LIN {X 0,Y 319.606,Z 333.555,A -85,B 0,C 180,E1 -15763.44,E2 -15763.44} C_VEL
LIN {X 0,Y 313.637,Z 316.329,A -85,B 0,C 180,E1 -15764.269,E2 -15764.269} C_VEL
LIN {X 0,Y 312.647,Z 311.538,A -85,B 0,C 180,E1 -15765.774,E2 -15765.774} C_VEL
LIN {X 0,Y 312.557,Z 311.55,A -85,B 0,C 180,E1 -15769.71,E2 -15769.71} C_VEL
LIN {X 0,Y 312.519,Z 311.556,A -85,B 0,C 180,E1 -15772.777,E2 -15772.777} C_VEL
LIN {X 0,Y 312.524,Z 311.552,A -85,B 0,C 180,E1 -15775.906,E2 -15775.906} C_VEL
LIN {X 0,Y 312.491,Z 311.556,A -85,B 0,C 180,E1 -15779.654,E2 -15779.654} C_VEL
LIN {X 0,Y 312.516,Z 311.553,A -85,B 0,C 180,E1 -15783.688,E2 -15783.688} C_VEL
LIN {X 0,Y 312.509,Z 311.554,A -85,B 0,C 180,E1 -15787.386,E2 -15787.386} C_VEL
LIN {X 0,Y 312.422,Z 311.565,A -85,B 0,C 180,E1 -15791.109,E2 -15791.109} C_VEL
LIN {X 0,Y 311.749,Z 311.65,A -85,B 0,C 180,E1 -15792.185,E2 -15792.185} C_VEL
LIN {X 0,Y 308.901,Z 312,A -85,B 0,C 180,E1 -15793.937,E2 -15793.937} C_VEL
LIN {X 0,Y 306.504,Z 312.305,A -85,B 0,C 180,E1 -15795.358,E2 -15795.358} C_VEL
LIN {X 0,Y 305.493,Z 312.428,A -85,B 0,C 180,E1 -15796.458,E2 -15796.458} C_VEL
LIN {X 0,Y 305.42,Z 312.437,A -85,B 0,C 180,E1 -15796.83,E2 -15796.83} C_VEL
LIN {X 0,Y 305.452,Z 312.431,A -85,B 0,C 180,E1 -15799.891,E2 -15799.891} C_VEL
LIN {X 0,Y 305.472,Z 312.433,A -85,B 0,C 180,E1 -15803.632,E2 -15803.632} C_VEL
LIN {X 0,Y 305.459,Z 312.432,A -85,B 0,C 180,E1 -15806.483,E2 -15806.483} C_VEL
LIN {X 0,Y 305.488,Z 312.425,A -85,B 0,C 180,E1 -15810.95,E2 -15810.95} C_VEL
LIN {X 0,Y 305.564,Z 312.421,A -85,B 0,C 180,E1 -15814.087,E2 -15814.087} C_VEL
LIN {X 0,Y 305.474,Z 312.427,A -85,B 0,C 180,E1 -15818.401,E2 -15818.401} C_VEL
LIN {X 0,Y 305.573,Z 312.415,A -85,B 0,C 180,E1 -15821.217,E2 -15821.217} C_VEL
LIN {X 0,Y 305.642,Z 312.411,A -85,B 0,C 180,E1 -15825.349,E2 -15825.349} C_VEL
LIN {X 0,Y 305.627,Z 312.408,A -85,B 0,C 180,E1 -15829.399,E2 -15829.399} C_VEL
LIN {X 0,Y 305.757,Z 312.396,A -85,B 0,C 180,E1 -15832.073,E2 -15832.073} C_VEL
LIN {X 0,Y 305.669,Z 312.408,A -85,B 0,C 180,E1 -15834.723,E2 -15834.723} C_VEL
LIN {X 0,Y 305.948,Z 312.37,A -85,B 0,C 180,E1 -15838.684,E2 -15838.684} C_VEL
LIN {X 0,Y 305.949,Z 312.366,A -85,B 0,C 180,E1 -15841.316,E2 -15841.316} C_VEL
LIN {X 0,Y 305.839,Z 312.389,A -85,B 0,C 180,E1 -15846.598,E2 -15846.598} C_VEL
LIN {X 0,Y 305.729,Z 312.396,A -85,B 0,C 180,E1 -15849.26,E2 -15849.26} C_VEL
LIN {X 0,Y 305.582,Z 312.417,A -85,B 0,C 180,E1 -15853.297,E2 -15853.297} C_VEL
LIN {X 0,Y 305.587,Z 312.417,A -85,B 0,C 180,E1 -15856.021,E2 -15856.021} C_VEL
LIN {X 0,Y 305.57,Z 312.42,A -85,B 0,C 180,E1 -15859.445,E2 -15859.445} C_VEL
LIN {X 0,Y 305.485,Z 312.434,A -85,B 0,C 180,E1 -15863.042,E2 -15863.042} C_VEL
LIN {X 0,Y 305.542,Z 312.422,A -85,B 0,C 180,E1 -15866.228,E2 -15866.228} C_VEL
LIN {X 0,Y 305.492,Z 312.434,A -85,B 0,C 180,E1 -15869.051,E2 -15869.051} C_VEL
LIN {X 0,Y 305.443,Z 312.436,A -85,B 0,C 180,E1 -15871.953,E2 -15871.953} C_VEL
LIN {X 0,Y 305.458,Z 312.438,A -85,B 0,C 180,E1 -15875.114,E2 -15875.114} C_VEL
LIN {X 0,Y 305.463,Z 312.434,A -85,B 0,C 180,E1 -15878.534,E2 -15878.534} C_VEL
LIN {X 0,Y 305.451,Z 312.435,A -85,B 0,C 180,E1 -15882.587,E2 -15882.587} C_VEL
LIN {X 0,Y 305.422,Z 312.438,A -85,B 0,C 180,E1 -15886.346,E2 -15886.346} C_VEL
LIN {X 0,Y 305.455,Z 312.437,A -85,B 0,C 180,E1 -15889.893,E2 -15889.893} C_VEL
LIN {X 0,Y 305.479,Z 312.435,A -85,B 0,C 180,E1 -15893.633,E2 -15893.633} C_VEL
LIN {X 0,Y 305.463,Z 312.435,A -85,B 0,C 180,E1 -15896.484,E2 -15896.484} C_VEL
LIN {X 0,Y 305.466,Z 312.471,A -85,B 0,C 180,E1 -15898.295,E2 -15898.295} C_VEL
LIN {X 0,Y 307.956,Z 324.046,A -85,B 0,C 180,E1 -15901.722,E2 -15901.722} C_VEL
LIN {X 0,Y 309.391,Z 332.337,A -85,B 0,C 180,E1 -15904.071,E2 -15904.071} C_VEL
LIN {X 0,Y 308.836,Z 337.527,A -85,B 0,C 180,E1 -15905.425,E2 -15905.425} C_VEL
LIN {X 0,Y 314.553,Z 379.23,A -85,B 0,C 180,E1 -15906.817,E2 -15906.817} C_VEL
LIN {X 0,Y 313.178,Z 446.148,A -85,B 0,C 180,E1 -15908.355,E2 -15908.355} C_VEL
LIN {X 0,Y 312.374,Z 459.427,A -85,B 0,C 180,E1 -15908.902,E2 -15908.902} C_VEL
LIN {X 0,Y 311.419,Z 472.21,A -85,B 0,C 180,E1 -15909.698,E2 -15909.698} C_VEL
LIN {X 0,Y 310.281,Z 483.534,A -85,B 0,C 180,E1 -15910.656,E2 -15910.656} C_VEL
LIN {X 0,Y 308.964,Z 495.25,A -85,B 0,C 180,E1 -15911.946,E2 -15911.946} C_VEL
LIN {X 0,Y 307.787,Z 505.776,A -85,B 0,C 180,E1 -15913.413,E2 -15913.413} C_VEL
LIN {X 0,Y 306.651,Z 515.269,A -85,B 0,C 180,E1 -15915.059,E2 -15915.059} C_VEL
LIN {X 0,Y 305.483,Z 524.396,A -85,B 0,C 180,E1 -15917.039,E2 -15917.039} C_VEL
LIN {X 0,Y 304.627,Z 531.743,A -85,B 0,C 180,E1 -15919.029,E2 -15919.029} C_VEL
LIN {X 0,Y 304.184,Z 536.708,A -85,B 0,C 180,E1 -15920.693,E2 -15920.693} C_VEL
LIN {X 0,Y 303.825,Z 541.519,A -85,B 0,C 180,E1 -15922.692,E2 -15922.692} C_VEL
LIN {X 0,Y 303.667,Z 545.193,A -85,B 0,C 180,E1 -15924.689,E2 -15924.689} C_VEL
LIN {X 0,Y 303.664,Z 547.088,A -85,B 0,C 180,E1 -15926.019,E2 -15926.019} C_VEL
LIN {X 0,Y 303.644,Z 548.512,A -85,B 0,C 180,E1 -15927.348,E2 -15927.348} C_VEL
LIN {X 0,Y 303.634,Z 549.517,A -85,B 0,C 180,E1 -15928.674,E2 -15928.674} C_VEL
LIN {X 0,Y 303.669,Z 550.131,A -85,B 0,C 180,E1 -15930.001,E2 -15930.001} C_VEL
LIN {X 0,Y 303.607,Z 550.351,A -85,B 0,C 180,E1 -15931.327,E2 -15931.327} C_VEL
LIN {X 0,Y 303.624,Z 550.145,A -85,B 0,C 180,E1 -15932.654,E2 -15932.654} C_VEL
LIN {X 0,Y 303.633,Z 549.536,A -85,B 0,C 180,E1 -15933.982,E2 -15933.982} C_VEL
LIN {X 0,Y 303.661,Z 548.281,A -85,B 0,C 180,E1 -15935.612,E2 -15935.612} C_VEL
LIN {X 0,Y 303.959,Z 545.322,A -85,B 0,C 180,E1 -15937.975,E2 -15937.975} C_VEL
LIN {X 0,Y 304.481,Z 541.759,A -85,B 0,C 180,E1 -15939.97,E2 -15939.97} C_VEL
LIN {X 0,Y 305.288,Z 537.11,A -85,B 0,C 180,E1 -15941.958,E2 -15941.958} C_VEL
LIN {X 0,Y 306.752,Z 530.122,A -85,B 0,C 180,E1 -15944.259,E2 -15944.259} C_VEL
LIN {X 0,Y 308.323,Z 522.727,A -85,B 0,C 180,E1 -15946.179,E2 -15946.179} C_VEL
LIN {X 0,Y 309.752,Z 514.917,A -85,B 0,C 180,E1 -15947.836,E2 -15947.836} C_VEL
LIN {X 0,Y 311.598,Z 505.596,A -85,B 0,C 180,E1 -15949.432,E2 -15949.432} C_VEL
LIN {X 0,Y 313.462,Z 495.268,A -85,B 0,C 180,E1 -15950.851,E2 -15950.851} C_VEL
LIN {X 0,Y 315.387,Z 483.82,A -85,B 0,C 180,E1 -15952.089,E2 -15952.089} C_VEL
LIN {X 0,Y 317.023,Z 471.841,A -85,B 0,C 180,E1 -15953.086,E2 -15953.086} C_VEL
LIN {X 0,Y 318.435,Z 458.547,A -85,B 0,C 180,E1 -15953.882,E2 -15953.882} C_VEL
LIN {X 0,Y 319.456,Z 445.222,A -85,B 0,C 180,E1 -15954.405,E2 -15954.405} C_VEL
LIN {X 0,Y 321.236,Z 381.833,A -85,B 0,C 180,E1 -15955.853,E2 -15955.853} C_VEL
LIN {X 0,Y 318.215,Z 363.674,A -85,B 0,C 180,E1 -15956.623,E2 -15956.623} C_VEL
LIN {X 0,Y 313.97,Z 343.479,A -85,B 0,C 180,E1 -15957.602,E2 -15957.602} C_VEL
LIN {X 0,Y 311.195,Z 336.716,A -85,B 0,C 180,E1 -15958.107,E2 -15958.107} C_VEL
LIN {X 0,Y 309.342,Z 328.013,A -85,B 0,C 180,E1 -15960.837,E2 -15960.837} C_VEL
LIN {X 0,Y 306.721,Z 317.256,A -85,B 0,C 180,E1 -15964.423,E2 -15964.423} C_VEL
LIN {X 0,Y 305.48,Z 312.435,A -85,B 0,C 180,E1 -15966.171,E2 -15966.171} C_VEL
LIN {X 0,Y 305.46,Z 312.434,A -85,B 0,C 180,E1 -15970.108,E2 -15970.108} C_VEL
LIN {X 0,Y 305.427,Z 312.441,A -85,B 0,C 180,E1 -15973.655,E2 -15973.655} C_VEL
LIN {X 0,Y 305.456,Z 312.433,A -85,B 0,C 180,E1 -15977.414,E2 -15977.414} C_VEL
LIN {X 0,Y 305.468,Z 312.433,A -85,B 0,C 180,E1 -15981.596,E2 -15981.596} C_VEL
LIN {X 0,Y 305.463,Z 312.434,A -85,B 0,C 180,E1 -15984.887,E2 -15984.887} C_VEL
LIN {X 0,Y 305.453,Z 312.435,A -85,B 0,C 180,E1 -15988.355,E2 -15988.355} C_VEL
LIN {X 0,Y 305.521,Z 312.428,A -85,B 0,C 180,E1 -15991.114,E2 -15991.114} C_VEL
LIN {X 0,Y 305.572,Z 312.418,A -85,B 0,C 180,E1 -15994.088,E2 -15994.088} C_VEL
LIN {X 0,Y 305.501,Z 312.427,A -85,B 0,C 180,E1 -15998.403,E2 -15998.403} C_VEL
LIN {X 0,Y 305.591,Z 312.412,A -85,B 0,C 180,E1 -16001.217,E2 -16001.217} C_VEL
LIN {X 0,Y 305.649,Z 312.403,A -85,B 0,C 180,E1 -16005.349,E2 -16005.349} C_VEL
LIN {X 0,Y 305.636,Z 312.404,A -85,B 0,C 180,E1 -16009.399,E2 -16009.399} C_VEL
LIN {X 0,Y 305.797,Z 312.39,A -85,B 0,C 180,E1 -16012.074,E2 -16012.074} C_VEL
LIN {X 0,Y 305.686,Z 312.393,A -85,B 0,C 180,E1 -16014.723,E2 -16014.723} C_VEL
LIN {X 0,Y 305.955,Z 312.358,A -85,B 0,C 180,E1 -16018.684,E2 -16018.684} C_VEL
LIN {X 0,Y 305.955,Z 312.368,A -85,B 0,C 180,E1 -16021.316,E2 -16021.316} C_VEL
LIN {X 0,Y 305.849,Z 312.379,A -85,B 0,C 180,E1 -16026.614,E2 -16026.614} C_VEL
LIN {X 0,Y 305.736,Z 312.396,A -85,B 0,C 180,E1 -16029.26,E2 -16029.26} C_VEL
LIN {X 0,Y 305.588,Z 312.415,A -85,B 0,C 180,E1 -16033.296,E2 -16033.296} C_VEL
LIN {X 0,Y 305.594,Z 312.414,A -85,B 0,C 180,E1 -16036.02,E2 -16036.02} C_VEL
LIN {X 0,Y 305.575,Z 312.418,A -85,B 0,C 180,E1 -16039.444,E2 -16039.444} C_VEL
LIN {X 0,Y 305.486,Z 312.431,A -85,B 0,C 180,E1 -16043.039,E2 -16043.039} C_VEL
LIN {X 0,Y 305.531,Z 312.423,A -85,B 0,C 180,E1 -16046.221,E2 -16046.221} C_VEL
LIN {X 0,Y 305.488,Z 312.426,A -85,B 0,C 180,E1 -16049.047,E2 -16049.047} C_VEL
LIN {X 0,Y 305.442,Z 312.429,A -85,B 0,C 180,E1 -16051.952,E2 -16051.952} C_VEL
LIN {X 0,Y 305.462,Z 312.429,A -85,B 0,C 180,E1 -16055.113,E2 -16055.113} C_VEL
LIN {X 0,Y 305.449,Z 312.435,A -85,B 0,C 180,E1 -16058.528,E2 -16058.528} C_VEL
LIN {X 0,Y 305.455,Z 312.433,A -85,B 0,C 180,E1 -16062.586,E2 -16062.586} C_VEL
LIN {X 0,Y 305.426,Z 312.439,A -85,B 0,C 180,E1 -16066.345,E2 -16066.345} C_VEL
LIN {X 0,Y 305.477,Z 312.557,A -85,B 0,C 180,E1 -16069.711,E2 -16069.711} C_VEL
LIN {X 0,Y 306.8,Z 317.441,A -85,B 0,C 180,E1 -16071.434,E2 -16071.434} C_VEL
LIN {X 0,Y 315.389,Z 334.724,A -85,B 0,C 180,E1 -16072.88,E2 -16072.88} C_VEL
LIN {X 0,Y 322.124,Z 350.394,A -85,B 0,C 180,E1 -16073.998,E2 -16073.998} C_VEL
LIN {X 0,Y 319.78,Z 424.71,A -85,B 0,C 180,E1 -16075.676,E2 -16075.676} C_VEL
LIN {X 0,Y 318.861,Z 438.142,A -85,B 0,C 180,E1 -16076.231,E2 -16076.231} C_VEL
LIN {X 0,Y 317.875,Z 450.412,A -85,B 0,C 180,E1 -16077.005,E2 -16077.005} C_VEL
LIN {X 0,Y 316.455,Z 462.001,A -85,B 0,C 180,E1 -16077.979,E2 -16077.979} C_VEL
LIN {X 0,Y 314.745,Z 473.836,A -85,B 0,C 180,E1 -16079.284,E2 -16079.284} C_VEL
LIN {X 0,Y 312.988,Z 484.195,A -85,B 0,C 180,E1 -16080.727,E2 -16080.727} C_VEL
LIN {X 0,Y 311.108,Z 493.835,A -85,B 0,C 180,E1 -16082.412,E2 -16082.412} C_VEL
LIN {X 0,Y 309.169,Z 502.926,A -85,B 0,C 180,E1 -16084.411,E2 -16084.411} C_VEL
LIN {X 0,Y 307.622,Z 510.346,A -85,B 0,C 180,E1 -16086.491,E2 -16086.491} C_VEL
LIN {X 0,Y 306.357,Z 515.897,A -85,B 0,C 180,E1 -16088.466,E2 -16088.466} C_VEL
LIN {X 0,Y 305.292,Z 520.731,A -85,B 0,C 180,E1 -16090.707,E2 -16090.707} C_VEL
LIN {X 0,Y 304.609,Z 523.698,A -85,B 0,C 180,E1 -16092.546,E2 -16092.546} C_VEL
LIN {X 0,Y 304.22,Z 525.341,A -85,B 0,C 180,E1 -16093.905,E2 -16093.905} C_VEL
LIN {X 0,Y 303.862,Z 527.186,A -85,B 0,C 180,E1 -16096.268,E2 -16096.268} C_VEL
LIN {X 0,Y 303.648,Z 527.726,A -85,B 0,C 180,E1 -16097.976,E2 -16097.976} C_VEL
LIN {X 0,Y 303.522,Z 527.294,A -85,B 0,C 180,E1 -16100.672,E2 -16100.672} C_VEL
LIN {X 0,Y 303.609,Z 526.451,A -85,B 0,C 180,E1 -16102.016,E2 -16102.016} C_VEL
LIN {X 0,Y 303.858,Z 524.443,A -85,B 0,C 180,E1 -16104.019,E2 -16104.019} C_VEL
LIN {X 0,Y 304.008,Z 521.468,A -85,B 0,C 180,E1 -16106.022,E2 -16106.022} C_VEL
LIN {X 0,Y 304.393,Z 517.456,A -85,B 0,C 180,E1 -16108.015,E2 -16108.015} C_VEL
LIN {X 0,Y 304.979,Z 511.297,A -85,B 0,C 180,E1 -16110.329,E2 -16110.329} C_VEL
LIN {X 0,Y 305.887,Z 504.58,A -85,B 0,C 180,E1 -16112.304,E2 -16112.304} C_VEL
LIN {X 0,Y 306.922,Z 496.259,A -85,B 0,C 180,E1 -16114.267,E2 -16114.267} C_VEL
LIN {X 0,Y 307.979,Z 487.688,A -85,B 0,C 180,E1 -16115.893,E2 -16115.893} C_VEL
LIN {X 0,Y 309.225,Z 477.138,A -85,B 0,C 180,E1 -16117.508,E2 -16117.508} C_VEL
LIN {X 0,Y 310.583,Z 466.616,A -85,B 0,C 180,E1 -16118.785,E2 -16118.785} C_VEL
LIN {X 0,Y 311.677,Z 455.001,A -85,B 0,C 180,E1 -16119.9,E2 -16119.9} C_VEL
LIN {X 0,Y 312.445,Z 442.998,A -85,B 0,C 180,E1 -16120.776,E2 -16120.776} C_VEL
LIN {X 0,Y 312.941,Z 430.888,A -85,B 0,C 180,E1 -16121.414,E2 -16121.414} C_VEL
LIN {X 0,Y 313.57,Z 419.55,A -85,B 0,C 180,E1 -16121.779,E2 -16121.779} C_VEL
LIN {X 0,Y 315.154,Z 346.424,A -85,B 0,C 180,E1 -16123.428,E2 -16123.428} C_VEL
LIN {X 0,Y 313.234,Z 335.967,A -85,B 0,C 180,E1 -16123.808,E2 -16123.808} C_VEL
LIN {X 0,Y 306.462,Z 316.608,A -85,B 0,C 180,E1 -16124.772,E2 -16124.772} C_VEL
LIN {X 0,Y 305.582,Z 312.42,A -85,B 0,C 180,E1 -16126.105,E2 -16126.105} C_VEL
LIN {X 0,Y 305.493,Z 312.433,A -85,B 0,C 180,E1 -16130.186,E2 -16130.186} C_VEL
LIN {X 0,Y 305.471,Z 312.435,A -85,B 0,C 180,E1 -16134.463,E2 -16134.463} C_VEL
LIN {X 0,Y 305.451,Z 312.433,A -85,B 0,C 180,E1 -16137.397,E2 -16137.397} C_VEL
LIN {X 0,Y 305.427,Z 312.439,A -85,B 0,C 180,E1 -16140.412,E2 -16140.412} C_VEL
LIN {X 0,Y 305.461,Z 312.433,A -85,B 0,C 180,E1 -16144.077,E2 -16144.077} C_VEL
LIN {X 0,Y 305.465,Z 312.436,A -85,B 0,C 180,E1 -16146.739,E2 -16146.739} C_VEL
LIN {X 0,Y 305.404,Z 312.441,A -85,B 0,C 180,E1 -16150.589,E2 -16150.589} C_VEL
LIN {X 0,Y 305.416,Z 312.435,A -85,B 0,C 180,E1 -16153.655,E2 -16153.655} C_VEL
LIN {X 0,Y 305.42,Z 312.437,A -85,B 0,C 180,E1 -16156.83,E2 -16156.83} C_VEL
LIN {X 0,Y 304.771,Z 312.52,A -85,B 0,C 180,E1 -16157.932,E2 -16157.932} C_VEL
LIN {X 0,Y 301.911,Z 312.873,A -85,B 0,C 180,E1 -16159.725,E2 -16159.725} C_VEL
LIN {X 0,Y 299.49,Z 313.175,A -85,B 0,C 180,E1 -16161.179,E2 -16161.179} C_VEL
LIN {X 0,Y 298.475,Z 313.299,A -85,B 0,C 180,E1 -16162.306,E2 -16162.306} C_VEL
LIN {X 0,Y 298.405,Z 313.308,A -85,B 0,C 180,E1 -16162.688,E2 -16162.688} C_VEL
LIN {X 0,Y 298.402,Z 313.315,A -85,B 0,C 180,E1 -16165.58,E2 -16165.58} C_VEL
LIN {X 0,Y 298.388,Z 313.31,A -85,B 0,C 180,E1 -16168.791,E2 -16168.791} C_VEL
LIN {X 0,Y 298.457,Z 313.306,A -85,B 0,C 180,E1 -16171.904,E2 -16171.904} C_VEL
LIN {X 0,Y 298.477,Z 313.303,A -85,B 0,C 180,E1 -16174.923,E2 -16174.923} C_VEL
LIN {X 0,Y 298.43,Z 313.305,A -85,B 0,C 180,E1 -16179.314,E2 -16179.314} C_VEL
LIN {X 0,Y 298.528,Z 313.297,A -85,B 0,C 180,E1 -16182.179,E2 -16182.179} C_VEL
LIN {X 0,Y 298.586,Z 313.289,A -85,B 0,C 180,E1 -16184.995,E2 -16184.995} C_VEL
LIN {X 0,Y 298.584,Z 313.284,A -85,B 0,C 180,E1 -16189.146,E2 -16189.146} C_VEL
LIN {X 0,Y 298.705,Z 313.272,A -85,B 0,C 180,E1 -16191.885,E2 -16191.885} C_VEL
LIN {X 0,Y 298.637,Z 313.284,A -85,B 0,C 180,E1 -16194.599,E2 -16194.599} C_VEL
LIN {X 0,Y 298.914,Z 313.246,A -85,B 0,C 180,E1 -16198.653,E2 -16198.653} C_VEL
LIN {X 0,Y 298.916,Z 313.241,A -85,B 0,C 180,E1 -16201.347,E2 -16201.347} C_VEL
LIN {X 0,Y 298.785,Z 313.266,A -85,B 0,C 180,E1 -16206.754,E2 -16206.754} C_VEL
LIN {X 0,Y 298.673,Z 313.274,A -85,B 0,C 180,E1 -16209.481,E2 -16209.481} C_VEL
LIN {X 0,Y 298.545,Z 313.292,A -85,B 0,C 180,E1 -16213.616,E2 -16213.616} C_VEL
LIN {X 0,Y 298.542,Z 313.297,A -85,B 0,C 180,E1 -16216.409,E2 -16216.409} C_VEL
LIN {X 0,Y 298.505,Z 313.299,A -85,B 0,C 180,E1 -16219.655,E2 -16219.655} C_VEL
LIN {X 0,Y 298.452,Z 313.307,A -85,B 0,C 180,E1 -16223.598,E2 -16223.598} C_VEL
LIN {X 0,Y 298.484,Z 313.303,A -85,B 0,C 180,E1 -16226.575,E2 -16226.575} C_VEL
LIN {X 0,Y 298.417,Z 313.311,A -85,B 0,C 180,E1 -16229.642,E2 -16229.642} C_VEL
LIN {X 0,Y 298.393,Z 313.316,A -85,B 0,C 180,E1 -16232.801,E2 -16232.801} C_VEL
LIN {X 0,Y 298.46,Z 313.307,A -85,B 0,C 180,E1 -16236.813,E2 -16236.813} C_VEL
LIN {X 0,Y 298.383,Z 313.318,A -85,B 0,C 180,E1 -16241.089,E2 -16241.089} C_VEL
LIN {X 0,Y 298.395,Z 313.316,A -85,B 0,C 180,E1 -16243.104,E2 -16243.104} C_VEL
LIN {X 0,Y 298.399,Z 313.314,A -85,B 0,C 180,E1 -16246.922,E2 -16246.922} C_VEL
LIN {X 0,Y 298.412,Z 313.312,A -85,B 0,C 180,E1 -16251.005,E2 -16251.005} C_VEL
LIN {X 0,Y 298.416,Z 313.315,A -85,B 0,C 180,E1 -16253.931,E2 -16253.931} C_VEL
LIN {X 0,Y 298.418,Z 313.421,A -85,B 0,C 180,E1 -16257.933,E2 -16257.933} C_VEL
LIN {X 0,Y 300.881,Z 324.79,A -85,B 0,C 180,E1 -16261.392,E2 -16261.392} C_VEL
LIN {X 0,Y 302.369,Z 333.039,A -85,B 0,C 180,E1 -16263.794,E2 -16263.794} C_VEL
LIN {X 0,Y 302.007,Z 337.242,A -85,B 0,C 180,E1 -16264.924,E2 -16264.924} C_VEL
LIN {X 0,Y 306.284,Z 368.116,A -85,B 0,C 180,E1 -16266,E2 -16266} C_VEL
LIN {X 0,Y 307.883,Z 380.76,A -85,B 0,C 180,E1 -16266.418,E2 -16266.418} C_VEL
LIN {X 0,Y 306.439,Z 445.861,A -85,B 0,C 180,E1 -16267.943,E2 -16267.943} C_VEL
LIN {X 0,Y 305.636,Z 459.154,A -85,B 0,C 180,E1 -16268.503,E2 -16268.503} C_VEL
LIN {X 0,Y 304.626,Z 471.934,A -85,B 0,C 180,E1 -16269.313,E2 -16269.313} C_VEL
LIN {X 0,Y 303.359,Z 484.06,A -85,B 0,C 180,E1 -16270.372,E2 -16270.372} C_VEL
LIN {X 0,Y 302.015,Z 495.633,A -85,B 0,C 180,E1 -16271.692,E2 -16271.692} C_VEL
LIN {X 0,Y 300.8,Z 506.072,A -85,B 0,C 180,E1 -16273.196,E2 -16273.196} C_VEL
LIN {X 0,Y 299.763,Z 514.583,A -85,B 0,C 180,E1 -16274.708,E2 -16274.708} C_VEL
LIN {X 0,Y 298.528,Z 523.787,A -85,B 0,C 180,E1 -16276.731,E2 -16276.731} C_VEL
LIN {X 0,Y 297.609,Z 531.193,A -85,B 0,C 180,E1 -16278.767,E2 -16278.767} C_VEL
LIN {X 0,Y 297.129,Z 536.212,A -85,B 0,C 180,E1 -16280.47,E2 -16280.47} C_VEL
LIN {X 0,Y 296.773,Z 541.075,A -85,B 0,C 180,E1 -16282.517,E2 -16282.517} C_VEL
LIN {X 0,Y 296.581,Z 544.794,A -85,B 0,C 180,E1 -16284.562,E2 -16284.562} C_VEL
LIN {X 0,Y 296.579,Z 546.713,A -85,B 0,C 180,E1 -16285.924,E2 -16285.924} C_VEL
LIN {X 0,Y 296.569,Z 548.178,A -85,B 0,C 180,E1 -16287.284,E2 -16287.284} C_VEL
LIN {X 0,Y 296.55,Z 549.203,A -85,B 0,C 180,E1 -16288.643,E2 -16288.643} C_VEL
LIN {X 0,Y 296.58,Z 549.836,A -85,B 0,C 180,E1 -16290.001,E2 -16290.001} C_VEL
LIN {X 0,Y 296.525,Z 550.077,A -85,B 0,C 180,E1 -16291.359,E2 -16291.359} C_VEL
LIN {X 0,Y 296.548,Z 549.91,A -85,B 0,C 180,E1 -16292.717,E2 -16292.717} C_VEL
LIN {X 0,Y 296.531,Z 549.32,A -85,B 0,C 180,E1 -16294.078,E2 -16294.078} C_VEL
LIN {X 0,Y 296.688,Z 546.98,A -85,B 0,C 180,E1 -16296.803,E2 -16296.803} C_VEL
LIN {X 0,Y 297.07,Z 544.113,A -85,B 0,C 180,E1 -16298.846,E2 -16298.846} C_VEL
LIN {X 0,Y 297.736,Z 540.237,A -85,B 0,C 180,E1 -16300.886,E2 -16300.886} C_VEL
LIN {X 0,Y 298.694,Z 535.255,A -85,B 0,C 180,E1 -16302.917,E2 -16302.917} C_VEL
LIN {X 0,Y 300.149,Z 529.018,A -85,B 0,C 180,E1 -16304.926,E2 -16304.926} C_VEL
LIN {X 0,Y 301.602,Z 521.824,A -85,B 0,C 180,E1 -16306.799,E2 -16306.799} C_VEL
LIN {X 0,Y 303.309,Z 513.533,A -85,B 0,C 180,E1 -16308.544,E2 -16308.544} C_VEL
LIN {X 0,Y 305.337,Z 503.735,A -85,B 0,C 180,E1 -16310.198,E2 -16310.198} C_VEL
LIN {X 0,Y 307.377,Z 493.078,A -85,B 0,C 180,E1 -16311.635,E2 -16311.635} C_VEL
LIN {X 0,Y 309.109,Z 482.78,A -85,B 0,C 180,E1 -16312.738,E2 -16312.738} C_VEL
LIN {X 0,Y 310.819,Z 470.479,A -85,B 0,C 180,E1 -16313.751,E2 -16313.751} C_VEL
LIN {X 0,Y 312.23,Z 457.564,A -85,B 0,C 180,E1 -16314.52,E2 -16314.52} C_VEL
LIN {X 0,Y 313.204,Z 445.032,A -85,B 0,C 180,E1 -16315.014,E2 -16315.014} C_VEL
LIN {X 0,Y 314.974,Z 382.045,A -85,B 0,C 180,E1 -16316.488,E2 -16316.488} C_VEL
LIN {X 0,Y 311.512,Z 361.958,A -85,B 0,C 180,E1 -16317.385,E2 -16317.385} C_VEL
LIN {X 0,Y 308.054,Z 346.009,A -85,B 0,C 180,E1 -16318.199,E2 -16318.199} C_VEL
LIN {X 0,Y 303.959,Z 336.373,A -85,B 0,C 180,E1 -16318.965,E2 -16318.965} C_VEL
LIN {X 0,Y 301.908,Z 327.151,A -85,B 0,C 180,E1 -16321.978,E2 -16321.978} C_VEL
LIN {X 0,Y 299.597,Z 317.673,A -85,B 0,C 180,E1 -16325.263,E2 -16325.263} C_VEL
LIN {X 0,Y 298.43,Z 313.311,A -85,B 0,C 180,E1 -16326.885,E2 -16326.885} C_VEL
LIN {X 0,Y 298.389,Z 313.318,A -85,B 0,C 180,E1 -16331.088,E2 -16331.088} C_VEL
LIN {X 0,Y 298.4,Z 313.316,A -85,B 0,C 180,E1 -16333.103,E2 -16333.103} C_VEL
LIN {X 0,Y 298.404,Z 313.311,A -85,B 0,C 180,E1 -16336.921,E2 -16336.921} C_VEL
LIN {X 0,Y 298.4,Z 313.315,A -85,B 0,C 180,E1 -16341.007,E2 -16341.007} C_VEL
LIN {X 0,Y 298.419,Z 313.31,A -85,B 0,C 180,E1 -16343.93,E2 -16343.93} C_VEL
LIN {X 0,Y 298.396,Z 313.313,A -85,B 0,C 180,E1 -16347.983,E2 -16347.983} C_VEL
LIN {X 0,Y 298.464,Z 313.305,A -85,B 0,C 180,E1 -16351.904,E2 -16351.904} C_VEL
LIN {X 0,Y 298.486,Z 313.304,A -85,B 0,C 180,E1 -16354.924,E2 -16354.924} C_VEL
LIN {X 0,Y 298.451,Z 313.311,A -85,B 0,C 180,E1 -16359.315,E2 -16359.315} C_VEL
LIN {X 0,Y 298.538,Z 313.293,A -85,B 0,C 180,E1 -16362.179,E2 -16362.179} C_VEL
LIN {X 0,Y 298.594,Z 313.283,A -85,B 0,C 180,E1 -16364.995,E2 -16364.995} C_VEL
LIN {X 0,Y 298.592,Z 313.284,A -85,B 0,C 180,E1 -16369.146,E2 -16369.146} C_VEL
LIN {X 0,Y 298.742,Z 313.27,A -85,B 0,C 180,E1 -16371.885,E2 -16371.885} C_VEL
LIN {X 0,Y 298.657,Z 313.269,A -85,B 0,C 180,E1 -16374.599,E2 -16374.599} C_VEL
LIN {X 0,Y 298.921,Z 313.234,A -85,B 0,C 180,E1 -16378.653,E2 -16378.653} C_VEL
LIN {X 0,Y 298.921,Z 313.244,A -85,B 0,C 180,E1 -16381.347,E2 -16381.347} C_VEL
LIN {X 0,Y 298.797,Z 313.257,A -85,B 0,C 180,E1 -16386.754,E2 -16386.754} C_VEL
LIN {X 0,Y 298.681,Z 313.275,A -85,B 0,C 180,E1 -16389.48,E2 -16389.48} C_VEL
LIN {X 0,Y 298.552,Z 313.292,A -85,B 0,C 180,E1 -16393.615,E2 -16393.615} C_VEL
LIN {X 0,Y 298.549,Z 313.289,A -85,B 0,C 180,E1 -16396.409,E2 -16396.409} C_VEL
LIN {X 0,Y 298.51,Z 313.298,A -85,B 0,C 180,E1 -16399.654,E2 -16399.654} C_VEL
LIN {X 0,Y 298.429,Z 313.307,A -85,B 0,C 180,E1 -16403.6,E2 -16403.6} C_VEL
LIN {X 0,Y 298.487,Z 313.303,A -85,B 0,C 180,E1 -16406.575,E2 -16406.575} C_VEL
LIN {X 0,Y 298.416,Z 313.31,A -85,B 0,C 180,E1 -16409.641,E2 -16409.641} C_VEL
LIN {X 0,Y 298.395,Z 313.311,A -85,B 0,C 180,E1 -16412.8,E2 -16412.8} C_VEL
LIN {X 0,Y 298.446,Z 313.308,A -85,B 0,C 180,E1 -16416.807,E2 -16416.807} C_VEL
LIN {X 0,Y 298.388,Z 313.315,A -85,B 0,C 180,E1 -16421.088,E2 -16421.088} C_VEL
LIN {X 0,Y 298.399,Z 313.313,A -85,B 0,C 180,E1 -16423.103,E2 -16423.103} C_VEL
LIN {X 0,Y 298.403,Z 313.313,A -85,B 0,C 180,E1 -16426.921,E2 -16426.921} C_VEL
LIN {X 0,Y 298.413,Z 313.413,A -85,B 0,C 180,E1 -16428.971,E2 -16428.971} C_VEL
LIN {X 0,Y 299.549,Z 317.672,A -85,B 0,C 180,E1 -16430.546,E2 -16430.546} C_VEL
LIN {X 0,Y 308.985,Z 336.297,A -85,B 0,C 180,E1 -16432.202,E2 -16432.202} C_VEL
LIN {X 0,Y 315.819,Z 351.992,A -85,B 0,C 180,E1 -16433.377,E2 -16433.377} C_VEL
LIN {X 0,Y 313.51,Z 425.536,A -85,B 0,C 180,E1 -16435.086,E2 -16435.086} C_VEL
LIN {X 0,Y 312.478,Z 439.554,A -85,B 0,C 180,E1 -16435.689,E2 -16435.689} C_VEL
LIN {X 0,Y 311.423,Z 451.94,A -85,B 0,C 180,E1 -16436.516,E2 -16436.516} C_VEL
LIN {X 0,Y 309.838,Z 464.077,A -85,B 0,C 180,E1 -16437.596,E2 -16437.596} C_VEL
LIN {X 0,Y 308.075,Z 475.573,A -85,B 0,C 180,E1 -16438.926,E2 -16438.926} C_VEL
LIN {X 0,Y 306.097,Z 486.207,A -85,B 0,C 180,E1 -16440.495,E2 -16440.495} C_VEL
LIN {X 0,Y 304.293,Z 495.016,A -85,B 0,C 180,E1 -16442.115,E2 -16442.115} C_VEL
LIN {X 0,Y 302.287,Z 503.946,A -85,B 0,C 180,E1 -16444.155,E2 -16444.155} C_VEL
LIN {X 0,Y 300.823,Z 510.469,A -85,B 0,C 180,E1 -16446.041,E2 -16446.041} C_VEL
LIN {X 0,Y 299.577,Z 515.794,A -85,B 0,C 180,E1 -16447.953,E2 -16447.953} C_VEL
LIN {X 0,Y 298.301,Z 521.104,A -85,B 0,C 180,E1 -16450.459,E2 -16450.459} C_VEL
LIN {X 0,Y 297.655,Z 523.762,A -85,B 0,C 180,E1 -16452.124,E2 -16452.124} C_VEL
LIN {X 0,Y 297.247,Z 525.443,A -85,B 0,C 180,E1 -16453.517,E2 -16453.517} C_VEL
LIN {X 0,Y 296.783,Z 527.483,A -85,B 0,C 180,E1 -16456.145,E2 -16456.145} C_VEL
LIN {X 0,Y 296.58,Z 527.976,A -85,B 0,C 180,E1 -16457.685,E2 -16457.685} C_VEL
LIN {X 0,Y 296.431,Z 527.616,A -85,B 0,C 180,E1 -16460.446,E2 -16460.446} C_VEL
LIN {X 0,Y 296.497,Z 526.842,A -85,B 0,C 180,E1 -16461.823,E2 -16461.823} C_VEL
LIN {X 0,Y 296.764,Z 524.653,A -85,B 0,C 180,E1 -16464.07,E2 -16464.07} C_VEL
LIN {X 0,Y 296.965,Z 520.775,A -85,B 0,C 180,E1 -16466.607,E2 -16466.607} C_VEL
LIN {X 0,Y 297.458,Z 516.474,A -85,B 0,C 180,E1 -16468.645,E2 -16468.645} C_VEL
LIN {X 0,Y 298.161,Z 509.992,A -85,B 0,C 180,E1 -16471.012,E2 -16471.012} C_VEL
LIN {X 0,Y 299.165,Z 502.859,A -85,B 0,C 180,E1 -16473.029,E2 -16473.029} C_VEL
LIN {X 0,Y 300.256,Z 494.019,A -85,B 0,C 180,E1 -16475.035,E2 -16475.035} C_VEL
LIN {X 0,Y 301.422,Z 484.945,A -85,B 0,C 180,E1 -16476.694,E2 -16476.694} C_VEL
LIN {X 0,Y 302.637,Z 474.881,A -85,B 0,C 180,E1 -16478.177,E2 -16478.177} C_VEL
LIN {X 0,Y 304.187,Z 463.632,A -85,B 0,C 180,E1 -16479.474,E2 -16479.474} C_VEL
LIN {X 0,Y 305.17,Z 451.13,A -85,B 0,C 180,E1 -16480.616,E2 -16480.616} C_VEL
LIN {X 0,Y 305.872,Z 438.235,A -85,B 0,C 180,E1 -16481.471,E2 -16481.471} C_VEL
LIN {X 0,Y 306.478,Z 426.662,A -85,B 0,C 180,E1 -16481.99,E2 -16481.99} C_VEL
LIN {X 0,Y 307.07,Z 412.17,A -85,B 0,C 180,E1 -16482.371,E2 -16482.371} C_VEL
LIN {X 0,Y 308.449,Z 347.055,A -85,B 0,C 180,E1 -16483.868,E2 -16483.868} C_VEL
LIN {X 0,Y 306.664,Z 337.666,A -85,B 0,C 180,E1 -16484.225,E2 -16484.225} C_VEL
LIN {X 0,Y 300.049,Z 319.06,A -85,B 0,C 180,E1 -16485.176,E2 -16485.176} C_VEL
LIN {X 0,Y 299.259,Z 316.788,A -85,B 0,C 180,E1 -16485.333,E2 -16485.333} C_VEL
LIN {X 0,Y 298.547,Z 313.297,A -85,B 0,C 180,E1 -16486.496,E2 -16486.496} C_VEL
LIN {X 0,Y 298.481,Z 313.304,A -85,B 0,C 180,E1 -16489.638,E2 -16489.638} C_VEL
LIN {X 0,Y 298.418,Z 313.309,A -85,B 0,C 180,E1 -16493.6,E2 -16493.6} C_VEL
LIN {X 0,Y 298.404,Z 313.313,A -85,B 0,C 180,E1 -16496.581,E2 -16496.581} C_VEL
LIN {X 0,Y 298.389,Z 313.312,A -85,B 0,C 180,E1 -16499.643,E2 -16499.643} C_VEL
LIN {X 0,Y 298.389,Z 313.318,A -85,B 0,C 180,E1 -16502.8,E2 -16502.8} C_VEL
LIN {X 0,Y 298.437,Z 313.312,A -85,B 0,C 180,E1 -16506.805,E2 -16506.805} C_VEL
LIN {X 0,Y 298.344,Z 313.324,A -85,B 0,C 180,E1 -16511.078,E2 -16511.078} C_VEL
LIN {X 0,Y 298.349,Z 313.318,A -85,B 0,C 180,E1 -16515.034,E2 -16515.034} C_VEL
LIN {X 0,Y 298.378,Z 313.316,A -85,B 0,C 180,E1 -16518.737,E2 -16518.737} C_VEL
LIN {X 0,Y 298.405,Z 313.308,A -85,B 0,C 180,E1 -16522.688,E2 -16522.688} C_VEL
LIN {X 0,Y 297.773,Z 313.393,A -85,B 0,C 180,E1 -16523.814,E2 -16523.814} C_VEL
LIN {X 0,Y 294.924,Z 313.747,A -85,B 0,C 180,E1 -16525.648,E2 -16525.648} C_VEL
LIN {X 0,Y 292.477,Z 314.052,A -85,B 0,C 180,E1 -16527.136,E2 -16527.136} C_VEL
LIN {X 0,Y 291.413,Z 314.178,A -85,B 0,C 180,E1 -16528.289,E2 -16528.289} C_VEL
LIN {X 0,Y 291.321,Z 314.187,A -85,B 0,C 180,E1 -16528.68,E2 -16528.68} C_VEL
LIN {X 0,Y 291.416,Z 314.18,A -85,B 0,C 180,E1 -16532.728,E2 -16532.728} C_VEL
LIN {X 0,Y 291.377,Z 314.186,A -85,B 0,C 180,E1 -16536.424,E2 -16536.424} C_VEL
LIN {X 0,Y 291.451,Z 314.173,A -85,B 0,C 180,E1 -16540.27,E2 -16540.27} C_VEL
LIN {X 0,Y 291.548,Z 314.166,A -85,B 0,C 180,E1 -16544.623,E2 -16544.623} C_VEL
LIN {X 0,Y 291.528,Z 314.162,A -85,B 0,C 180,E1 -16548.88,E2 -16548.88} C_VEL
LIN {X 0,Y 291.656,Z 314.148,A -85,B 0,C 180,E1 -16551.687,E2 -16551.687} C_VEL
LIN {X 0,Y 291.606,Z 314.161,A -85,B 0,C 180,E1 -16554.468,E2 -16554.468} C_VEL
LIN {X 0,Y 291.881,Z 314.121,A -85,B 0,C 180,E1 -16558.62,E2 -16558.62} C_VEL
LIN {X 0,Y 291.882,Z 314.117,A -85,B 0,C 180,E1 -16561.38,E2 -16561.38} C_VEL
LIN {X 0,Y 291.734,Z 314.143,A -85,B 0,C 180,E1 -16566.918,E2 -16566.918} C_VEL
LIN {X 0,Y 291.622,Z 314.151,A -85,B 0,C 180,E1 -16569.712,E2 -16569.712} C_VEL
LIN {X 0,Y 291.515,Z 314.168,A -85,B 0,C 180,E1 -16573.951,E2 -16573.951} C_VEL
LIN {X 0,Y 291.48,Z 314.178,A -85,B 0,C 180,E1 -16576.818,E2 -16576.818} C_VEL
LIN {X 0,Y 291.445,Z 314.179,A -85,B 0,C 180,E1 -16579.876,E2 -16579.876} C_VEL
LIN {X 0,Y 291.395,Z 314.185,A -85,B 0,C 180,E1 -16584.206,E2 -16584.206} C_VEL
LIN {X 0,Y 291.417,Z 314.186,A -85,B 0,C 180,E1 -16587.272,E2 -16587.272} C_VEL
LIN {X 0,Y 291.335,Z 314.192,A -85,B 0,C 180,E1 -16590.437,E2 -16590.437} C_VEL
LIN {X 0,Y 291.341,Z 314.194,A -85,B 0,C 180,E1 -16593.699,E2 -16593.699} C_VEL
LIN {X 0,Y 291.39,Z 314.19,A -85,B 0,C 180,E1 -16597.26,E2 -16597.26} C_VEL
LIN {X 0,Y 291.33,Z 314.194,A -85,B 0,C 180,E1 -16600.643,E2 -16600.643} C_VEL
LIN {X 0,Y 291.286,Z 314.199,A -85,B 0,C 180,E1 -16604.403,E2 -16604.403} C_VEL
LIN {X 0,Y 291.323,Z 314.195,A -85,B 0,C 180,E1 -16608.406,E2 -16608.406} C_VEL
LIN {X 0,Y 291.361,Z 314.191,A -85,B 0,C 180,E1 -16611.161,E2 -16611.161} C_VEL
LIN {X 0,Y 291.359,Z 314.192,A -85,B 0,C 180,E1 -16614.627,E2 -16614.627} C_VEL
LIN {X 0,Y 291.36,Z 314.228,A -85,B 0,C 180,E1 -16617.512,E2 -16617.512} C_VEL
LIN {X 0,Y 293.82,Z 325.474,A -85,B 0,C 180,E1 -16621.03,E2 -16621.03} C_VEL
LIN {X 0,Y 295.342,Z 333.736,A -85,B 0,C 180,E1 -16623.503,E2 -16623.503} C_VEL
LIN {X 0,Y 295.209,Z 336.969,A -85,B 0,C 180,E1 -16624.404,E2 -16624.404} C_VEL
LIN {X 0,Y 299.64,Z 368.824,A -85,B 0,C 180,E1 -16625.553,E2 -16625.553} C_VEL
LIN {X 0,Y 301.199,Z 381.297,A -85,B 0,C 180,E1 -16625.975,E2 -16625.975} C_VEL
LIN {X 0,Y 299.721,Z 445.576,A -85,B 0,C 180,E1 -16627.512,E2 -16627.512} C_VEL
LIN {X 0,Y 298.901,Z 458.878,A -85,B 0,C 180,E1 -16628.084,E2 -16628.084} C_VEL
LIN {X 0,Y 297.859,Z 471.662,A -85,B 0,C 180,E1 -16628.912,E2 -16628.912} C_VEL
LIN {X 0,Y 296.662,Z 482.995,A -85,B 0,C 180,E1 -16629.91,E2 -16629.91} C_VEL
LIN {X 0,Y 295.206,Z 494.707,A -85,B 0,C 180,E1 -16631.254,E2 -16631.254} C_VEL
LIN {X 0,Y 293.948,Z 505.259,A -85,B 0,C 180,E1 -16632.791,E2 -16632.791} C_VEL
LIN {X 0,Y 292.844,Z 514.092,A -85,B 0,C 180,E1 -16634.381,E2 -16634.381} C_VEL
LIN {X 0,Y 291.819,Z 521.799,A -85,B 0,C 180,E1 -16636.065,E2 -16636.065} C_VEL
LIN {X 0,Y 290.715,Z 529.512,A -85,B 0,C 180,E1 -16638.143,E2 -16638.143} C_VEL
LIN {X 0,Y 290.096,Z 535.717,A -85,B 0,C 180,E1 -16640.237,E2 -16640.237} C_VEL
LIN {X 0,Y 289.703,Z 540.629,A -85,B 0,C 180,E1 -16642.333,E2 -16642.333} C_VEL
LIN {X 0,Y 289.517,Z 544.396,A -85,B 0,C 180,E1 -16644.429,E2 -16644.429} C_VEL
LIN {X 0,Y 289.478,Z 546.335,A -85,B 0,C 180,E1 -16645.824,E2 -16645.824} C_VEL
LIN {X 0,Y 289.495,Z 547.841,A -85,B 0,C 180,E1 -16647.218,E2 -16647.218} C_VEL
LIN {X 0,Y 289.469,Z 548.888,A -85,B 0,C 180,E1 -16648.61,E2 -16648.61} C_VEL
LIN {X 0,Y 289.495,Z 549.542,A -85,B 0,C 180,E1 -16650.001,E2 -16650.001} C_VEL
LIN {X 0,Y 289.445,Z 549.803,A -85,B 0,C 180,E1 -16651.392,E2 -16651.392} C_VEL
LIN {X 0,Y 289.474,Z 549.671,A -85,B 0,C 180,E1 -16652.784,E2 -16652.784} C_VEL
LIN {X 0,Y 289.481,Z 548.15,A -85,B 0,C 180,E1 -16655.574,E2 -16655.574} C_VEL
LIN {X 0,Y 289.86,Z 545.052,A -85,B 0,C 180,E1 -16658.366,E2 -16658.366} C_VEL
LIN {X 0,Y 290.461,Z 541.568,A -85,B 0,C 180,E1 -16660.456,E2 -16660.456} C_VEL
LIN {X 0,Y 291.341,Z 537.016,A -85,B 0,C 180,E1 -16662.54,E2 -16662.54} C_VEL
LIN {X 0,Y 293,Z 530.153,A -85,B 0,C 180,E1 -16664.943,E2 -16664.943} C_VEL
LIN {X 0,Y 294.703,Z 522.347,A -85,B 0,C 180,E1 -16667.09,E2 -16667.09} C_VEL
LIN {X 0,Y 296.612,Z 513.551,A -85,B 0,C 180,E1 -16669.014,E2 -16669.014} C_VEL
LIN {X 0,Y 298.912,Z 502.961,A -85,B 0,C 180,E1 -16670.832,E2 -16670.832} C_VEL
LIN {X 0,Y 301.082,Z 492.195,A -85,B 0,C 180,E1 -16672.292,E2 -16672.292} C_VEL
LIN {X 0,Y 302.881,Z 481.721,A -85,B 0,C 180,E1 -16673.414,E2 -16673.414} C_VEL
LIN {X 0,Y 304.634,Z 469.147,A -85,B 0,C 180,E1 -16674.446,E2 -16674.446} C_VEL
LIN {X 0,Y 306.145,Z 455.844,A -85,B 0,C 180,E1 -16675.223,E2 -16675.223} C_VEL
LIN {X 0,Y 307.079,Z 443.499,A -85,B 0,C 180,E1 -16675.685,E2 -16675.685} C_VEL
LIN {X 0,Y 308.831,Z 383.174,A -85,B 0,C 180,E1 -16677.117,E2 -16677.117} C_VEL
LIN {X 0,Y 305.402,Z 362.998,A -85,B 0,C 180,E1 -16678.044,E2 -16678.044} C_VEL
LIN {X 0,Y 302.308,Z 348.742,A -85,B 0,C 180,E1 -16678.799,E2 -16678.799} C_VEL
LIN {X 0,Y 296.764,Z 336.037,A -85,B 0,C 180,E1 -16679.867,E2 -16679.867} C_VEL
LIN {X 0,Y 294.389,Z 325.914,A -85,B 0,C 180,E1 -16683.325,E2 -16683.325} C_VEL
LIN {X 0,Y 292.126,Z 317.085,A -85,B 0,C 180,E1 -16686.544,E2 -16686.544} C_VEL
LIN {X 0,Y 291.364,Z 314.193,A -85,B 0,C 180,E1 -16687.665,E2 -16687.665} C_VEL
LIN {X 0,Y 291.334,Z 314.194,A -85,B 0,C 180,E1 -16690.643,E2 -16690.643} C_VEL
LIN {X 0,Y 291.292,Z 314.198,A -85,B 0,C 180,E1 -16694.402,E2 -16694.402} C_VEL
LIN {X 0,Y 291.328,Z 314.196,A -85,B 0,C 180,E1 -16698.404,E2 -16698.404} C_VEL
LIN {X 0,Y 291.349,Z 314.194,A -85,B 0,C 180,E1 -16701.157,E2 -16701.157} C_VEL
LIN {X 0,Y 291.362,Z 314.192,A -85,B 0,C 180,E1 -16704.626,E2 -16704.626} C_VEL
LIN {X 0,Y 291.373,Z 314.188,A -85,B 0,C 180,E1 -16707.951,E2 -16707.951} C_VEL
LIN {X 0,Y 291.384,Z 314.19,A -85,B 0,C 180,E1 -16711.158,E2 -16711.158} C_VEL
LIN {X 0,Y 291.417,Z 314.181,A -85,B 0,C 180,E1 -16714.272,E2 -16714.272} C_VEL
LIN {X 0,Y 291.382,Z 314.182,A -85,B 0,C 180,E1 -16717.299,E2 -16717.299} C_VEL
LIN {X 0,Y 291.459,Z 314.175,A -85,B 0,C 180,E1 -16720.27,E2 -16720.27} C_VEL
LIN {X 0,Y 291.556,Z 314.162,A -85,B 0,C 180,E1 -16724.624,E2 -16724.624} C_VEL
LIN {X 0,Y 291.536,Z 314.164,A -85,B 0,C 180,E1 -16728.88,E2 -16728.88} C_VEL
LIN {X 0,Y 291.688,Z 314.146,A -85,B 0,C 180,E1 -16731.688,E2 -16731.688} C_VEL
LIN {X 0,Y 291.627,Z 314.144,A -85,B 0,C 180,E1 -16734.468,E2 -16734.468} C_VEL
LIN {X 0,Y 291.888,Z 314.11,A -85,B 0,C 180,E1 -16738.62,E2 -16738.62} C_VEL
LIN {X 0,Y 291.888,Z 314.12,A -85,B 0,C 180,E1 -16741.38,E2 -16741.38} C_VEL
LIN {X 0,Y 291.746,Z 314.134,A -85,B 0,C 180,E1 -16746.918,E2 -16746.918} C_VEL
LIN {X 0,Y 291.629,Z 314.154,A -85,B 0,C 180,E1 -16749.712,E2 -16749.712} C_VEL
LIN {X 0,Y 291.522,Z 314.169,A -85,B 0,C 180,E1 -16753.95,E2 -16753.95} C_VEL
LIN {X 0,Y 291.487,Z 314.169,A -85,B 0,C 180,E1 -16756.818,E2 -16756.818} C_VEL
LIN {X 0,Y 291.451,Z 314.178,A -85,B 0,C 180,E1 -16759.875,E2 -16759.875} C_VEL
LIN {X 0,Y 291.383,Z 314.182,A -85,B 0,C 180,E1 -16764.207,E2 -16764.207} C_VEL
LIN {X 0,Y 291.42,Z 314.178,A -85,B 0,C 180,E1 -16767.272,E2 -16767.272} C_VEL
LIN {X 0,Y 291.334,Z 314.193,A -85,B 0,C 180,E1 -16770.437,E2 -16770.437} C_VEL
LIN {X 0,Y 291.344,Z 314.19,A -85,B 0,C 180,E1 -16773.698,E2 -16773.698} C_VEL
LIN {X 0,Y 291.376,Z 314.185,A -85,B 0,C 180,E1 -16777.254,E2 -16777.254} C_VEL
LIN {X 0,Y 291.333,Z 314.191,A -85,B 0,C 180,E1 -16780.642,E2 -16780.642} C_VEL
LIN {X 0,Y 291.291,Z 314.199,A -85,B 0,C 180,E1 -16784.402,E2 -16784.402} C_VEL
LIN {X 0,Y 291.358,Z 314.33,A -85,B 0,C 180,E1 -16788.207,E2 -16788.207} C_VEL
LIN {X 0,Y 292.364,Z 318.041,A -85,B 0,C 180,E1 -16789.615,E2 -16789.615} C_VEL
LIN {X 0,Y 302.041,Z 336.62,A -85,B 0,C 180,E1 -16791.388,E2 -16791.388} C_VEL
LIN {X 0,Y 309.461,Z 353.333,A -85,B 0,C 180,E1 -16792.713,E2 -16792.713} C_VEL
LIN {X 0,Y 309.786,Z 354.212,A -85,B 0,C 180,E1 -16792.773,E2 -16792.773} C_VEL
LIN {X 0,Y 307.354,Z 425.199,A -85,B 0,C 180,E1 -16794.433,E2 -16794.433} C_VEL
LIN {X 0,Y 306.374,Z 438.644,A -85,B 0,C 180,E1 -16795.006,E2 -16795.006} C_VEL
LIN {X 0,Y 305.315,Z 450.474,A -85,B 0,C 180,E1 -16795.774,E2 -16795.774} C_VEL
LIN {X 0,Y 303.666,Z 462.909,A -85,B 0,C 180,E1 -16796.854,E2 -16796.854} C_VEL
LIN {X 0,Y 301.814,Z 474.67,A -85,B 0,C 180,E1 -16798.207,E2 -16798.207} C_VEL
LIN {X 0,Y 299.991,Z 484.433,A -85,B 0,C 180,E1 -16799.619,E2 -16799.619} C_VEL
LIN {X 0,Y 298.209,Z 492.962,A -85,B 0,C 180,E1 -16801.135,E2 -16801.135} C_VEL
LIN {X 0,Y 296.392,Z 500.837,A -85,B 0,C 180,E1 -16802.841,E2 -16802.841} C_VEL
LIN {X 0,Y 294.821,Z 507.429,A -85,B 0,C 180,E1 -16804.59,E2 -16804.59} C_VEL
LIN {X 0,Y 293.295,Z 513.835,A -85,B 0,C 180,E1 -16806.71,E2 -16806.71} C_VEL
LIN {X 0,Y 291.978,Z 518.882,A -85,B 0,C 180,E1 -16808.835,E2 -16808.835} C_VEL
LIN {X 0,Y 291.001,Z 522.749,A -85,B 0,C 180,E1 -16810.971,E2 -16810.971} C_VEL
LIN {X 0,Y 290.278,Z 525.546,A -85,B 0,C 180,E1 -16813.109,E2 -16813.109} C_VEL
LIN {X 0,Y 289.943,Z 526.849,A -85,B 0,C 180,E1 -16814.536,E2 -16814.536} C_VEL
LIN {X 0,Y 289.715,Z 527.775,A -85,B 0,C 180,E1 -16816.008,E2 -16816.008} C_VEL
LIN {X 0,Y 289.514,Z 528.226,A -85,B 0,C 180,E1 -16817.38,E2 -16817.38} C_VEL
LIN {X 0,Y 289.336,Z 527.937,A -85,B 0,C 180,E1 -16820.21,E2 -16820.21} C_VEL
LIN {X 0,Y 289.408,Z 527.21,A -85,B 0,C 180,E1 -16821.621,E2 -16821.621} C_VEL
LIN {X 0,Y 289.674,Z 524.873,A -85,B 0,C 180,E1 -16824.116,E2 -16824.116} C_VEL
LIN {X 0,Y 289.878,Z 521.317,A -85,B 0,C 180,E1 -16826.524,E2 -16826.524} C_VEL
LIN {X 0,Y 290.37,Z 517.098,A -85,B 0,C 180,E1 -16828.612,E2 -16828.612} C_VEL
LIN {X 0,Y 291.059,Z 510.716,A -85,B 0,C 180,E1 -16831.037,E2 -16831.037} C_VEL
LIN {X 0,Y 292.095,Z 503.727,A -85,B 0,C 180,E1 -16833.103,E2 -16833.103} C_VEL
LIN {X 0,Y 293.216,Z 495.008,A -85,B 0,C 180,E1 -16835.156,E2 -16835.156} C_VEL
LIN {X 0,Y 294.539,Z 485.107,A -85,B 0,C 180,E1 -16837.023,E2 -16837.023} C_VEL
LIN {X 0,Y 295.806,Z 475.009,A -85,B 0,C 180,E1 -16838.539,E2 -16838.539} C_VEL
LIN {X 0,Y 297.405,Z 463.727,A -85,B 0,C 180,E1 -16839.864,E2 -16839.864} C_VEL
LIN {X 0,Y 298.43,Z 451.168,A -85,B 0,C 180,E1 -16841.03,E2 -16841.03} C_VEL
LIN {X 0,Y 299.149,Z 438.172,A -85,B 0,C 180,E1 -16841.905,E2 -16841.905} C_VEL
LIN {X 0,Y 299.796,Z 426.341,A -85,B 0,C 180,E1 -16842.437,E2 -16842.437} C_VEL
LIN {X 0,Y 300.599,Z 403.812,A -85,B 0,C 180,E1 -16843.004,E2 -16843.004} C_VEL
LIN {X 0,Y 301.867,Z 348.374,A -85,B 0,C 180,E1 -16844.302,E2 -16844.302} C_VEL
LIN {X 0,Y 300.259,Z 339.823,A -85,B 0,C 180,E1 -16844.635,E2 -16844.635} C_VEL
LIN {X 0,Y 293.782,Z 321.655,A -85,B 0,C 180,E1 -16845.596,E2 -16845.596} C_VEL
LIN {X 0,Y 292.146,Z 317.146,A -85,B 0,C 180,E1 -16845.859,E2 -16845.859} C_VEL
LIN {X 0,Y 291.491,Z 314.174,A -85,B 0,C 180,E1 -16846.907,E2 -16846.907} C_VEL
LIN {X 0,Y 291.422,Z 314.184,A -85,B 0,C 180,E1 -16849.859,E2 -16849.859} C_VEL
LIN {X 0,Y 291.357,Z 314.191,A -85,B 0,C 180,E1 -16854.208,E2 -16854.208} C_VEL
LIN {X 0,Y 291.349,Z 314.19,A -85,B 0,C 180,E1 -16857.278,E2 -16857.278} C_VEL
LIN {X 0,Y 291.315,Z 314.197,A -85,B 0,C 180,E1 -16860.438,E2 -16860.438} C_VEL
LIN {X 0,Y 291.34,Z 314.192,A -85,B 0,C 180,E1 -16863.698,E2 -16863.698} C_VEL
LIN {X 0,Y 291.364,Z 314.189,A -85,B 0,C 180,E1 -16867.251,E2 -16867.251} C_VEL
LIN {X 0,Y 291.295,Z 314.199,A -85,B 0,C 180,E1 -16870.647,E2 -16870.647} C_VEL
LIN {X 0,Y 291.276,Z 314.195,A -85,B 0,C 180,E1 -16874.403,E2 -16874.403} C_VEL
LIN {X 0,Y 291.32,Z 314.193,A -85,B 0,C 180,E1 -16878.404,E2 -16878.404} C_VEL
LIN {X 0,Y 291.338,Z 314.19,A -85,B 0,C 180,E1 -16881.156,E2 -16881.156} C_VEL
LIN {X 0,Y 291.354,Z 314.189,A -85,B 0,C 180,E1 -16884.625,E2 -16884.625} C_VEL
LIN {X 0,Y 291.321,Z 314.187,A -85,B 0,C 180,E1 -16888.68,E2 -16888.68} C_VEL
LIN {X 0,Y 290.64,Z 314.275,A -85,B 0,C 180,E1 -16889.836,E2 -16889.836} C_VEL
LIN {X 0,Y 287.798,Z 314.633,A -85,B 0,C 180,E1 -16891.718,E2 -16891.718} C_VEL
LIN {X 0,Y 285.408,Z 314.931,A -85,B 0,C 180,E1 -16893.246,E2 -16893.246} C_VEL
LIN {X 0,Y 284.397,Z 315.057,A -85,B 0,C 180,E1 -16894.43,E2 -16894.43} C_VEL
LIN {X 0,Y 284.323,Z 315.065,A -85,B 0,C 180,E1 -16894.83,E2 -16894.83} C_VEL
LIN {X 0,Y 284.312,Z 315.062,A -85,B 0,C 180,E1 -16898.236,E2 -16898.236} C_VEL
LIN {X 0,Y 284.392,Z 315.052,A -85,B 0,C 180,E1 -16901.261,E2 -16901.261} C_VEL
LIN {X 0,Y 284.485,Z 315.047,A -85,B 0,C 180,E1 -16904.459,E2 -16904.459} C_VEL
LIN {X 0,Y 284.48,Z 315.04,A -85,B 0,C 180,E1 -16908.601,E2 -16908.601} C_VEL
LIN {X 0,Y 284.611,Z 315.024,A -85,B 0,C 180,E1 -16911.48,E2 -16911.48} C_VEL
LIN {X 0,Y 284.575,Z 315.038,A -85,B 0,C 180,E1 -16914.331,E2 -16914.331} C_VEL
LIN {X 0,Y 284.847,Z 314.997,A -85,B 0,C 180,E1 -16918.586,E2 -16918.586} C_VEL
LIN {X 0,Y 284.848,Z 314.992,A -85,B 0,C 180,E1 -16921.414,E2 -16921.414} C_VEL
LIN {X 0,Y 284.687,Z 315.02,A -85,B 0,C 180,E1 -16927.091,E2 -16927.091} C_VEL
LIN {X 0,Y 284.56,Z 315.031,A -85,B 0,C 180,E1 -16929.956,E2 -16929.956} C_VEL
LIN {X 0,Y 284.471,Z 315.047,A -85,B 0,C 180,E1 -16934.304,E2 -16934.304} C_VEL
LIN {X 0,Y 284.419,Z 315.054,A -85,B 0,C 180,E1 -16937.249,E2 -16937.249} C_VEL
LIN {X 0,Y 284.373,Z 315.06,A -85,B 0,C 180,E1 -16940.243,E2 -16940.243} C_VEL
LIN {X 0,Y 284.363,Z 315.061,A -85,B 0,C 180,E1 -16943.876,E2 -16943.876} C_VEL
LIN {X 0,Y 284.392,Z 315.062,A -85,B 0,C 180,E1 -16947.175,E2 -16947.175} C_VEL
LIN {X 0,Y 284.293,Z 315.075,A -85,B 0,C 180,E1 -16951.275,E2 -16951.275} C_VEL
LIN {X 0,Y 284.357,Z 315.067,A -85,B 0,C 180,E1 -16955.355,E2 -16955.355} C_VEL
LIN {X 0,Y 284.319,Z 315.068,A -85,B 0,C 180,E1 -16958.168,E2 -16958.168} C_VEL
LIN {X 0,Y 284.265,Z 315.075,A -85,B 0,C 180,E1 -16962.125,E2 -16962.125} C_VEL
LIN {X 0,Y 284.252,Z 315.076,A -85,B 0,C 180,E1 -16966.19,E2 -16966.19} C_VEL
LIN {X 0,Y 284.304,Z 315.071,A -85,B 0,C 180,E1 -16970.025,E2 -16970.025} C_VEL
LIN {X 0,Y 284.332,Z 315.07,A -85,B 0,C 180,E1 -16973.616,E2 -16973.616} C_VEL
LIN {X 0,Y 284.36,Z 315.205,A -85,B 0,C 180,E1 -16977.126,E2 -16977.126} C_VEL
LIN {X 0,Y 286.964,Z 327.268,A -85,B 0,C 180,E1 -16980.999,E2 -16980.999} C_VEL
LIN {X 0,Y 288.457,Z 335.787,A -85,B 0,C 180,E1 -16983.601,E2 -16983.601} C_VEL
LIN {X 0,Y 288.439,Z 336.628,A -85,B 0,C 180,E1 -16983.842,E2 -16983.842} C_VEL
LIN {X 0,Y 292.546,Z 365.93,A -85,B 0,C 180,E1 -16984.958,E2 -16984.958} C_VEL
LIN {X 0,Y 294.503,Z 382.97,A -85,B 0,C 180,E1 -16985.542,E2 -16985.542} C_VEL
LIN {X 0,Y 293.02,Z 445.276,A -85,B 0,C 180,E1 -16987.065,E2 -16987.065} C_VEL
LIN {X 0,Y 292.176,Z 458.544,A -85,B 0,C 180,E1 -16987.646,E2 -16987.646} C_VEL
LIN {X 0,Y 291.11,Z 471.351,A -85,B 0,C 180,E1 -16988.492,E2 -16988.492} C_VEL
LIN {X 0,Y 289.768,Z 483.498,A -85,B 0,C 180,E1 -16989.596,E2 -16989.596} C_VEL
LIN {X 0,Y 288.273,Z 495.072,A -85,B 0,C 180,E1 -16990.97,E2 -16990.97} C_VEL
LIN {X 0,Y 286.978,Z 505.518,A -85,B 0,C 180,E1 -16992.544,E2 -16992.544} C_VEL
LIN {X 0,Y 285.755,Z 514.874,A -85,B 0,C 180,E1 -16994.305,E2 -16994.305} C_VEL
LIN {X 0,Y 284.439,Z 523.934,A -85,B 0,C 180,E1 -16996.425,E2 -16996.425} C_VEL
LIN {X 0,Y 283.459,Z 531.222,A -85,B 0,C 180,E1 -16998.56,E2 -16998.56} C_VEL
LIN {X 0,Y 282.885,Z 537.036,A -85,B 0,C 180,E1 -17000.708,E2 -17000.708} C_VEL
LIN {X 0,Y 282.551,Z 541.598,A -85,B 0,C 180,E1 -17002.857,E2 -17002.857} C_VEL
LIN {X 0,Y 282.415,Z 544.334,A -85,B 0,C 180,E1 -17004.513,E2 -17004.513} C_VEL
LIN {X 0,Y 282.422,Z 547.497,A -85,B 0,C 180,E1 -17007.148,E2 -17007.148} C_VEL
LIN {X 0,Y 282.39,Z 548.574,A -85,B 0,C 180,E1 -17008.575,E2 -17008.575} C_VEL
LIN {X 0,Y 282.412,Z 549.247,A -85,B 0,C 180,E1 -17010.001,E2 -17010.001} C_VEL
LIN {X 0,Y 282.367,Z 549.528,A -85,B 0,C 180,E1 -17011.427,E2 -17011.427} C_VEL
LIN {X 0,Y 282.378,Z 549.423,A -85,B 0,C 180,E1 -17012.854,E2 -17012.854} C_VEL
LIN {X 0,Y 282.376,Z 548.205,A -85,B 0,C 180,E1 -17015.403,E2 -17015.403} C_VEL
LIN {X 0,Y 282.552,Z 546.631,A -85,B 0,C 180,E1 -17017.145,E2 -17017.145} C_VEL
LIN {X 0,Y 282.993,Z 543.851,A -85,B 0,C 180,E1 -17019.29,E2 -17019.29} C_VEL
LIN {X 0,Y 283.756,Z 540.069,A -85,B 0,C 180,E1 -17021.429,E2 -17021.429} C_VEL
LIN {X 0,Y 284.828,Z 535.187,A -85,B 0,C 180,E1 -17023.557,E2 -17023.557} C_VEL
LIN {X 0,Y 286.416,Z 529.061,A -85,B 0,C 180,E1 -17025.66,E2 -17025.66} C_VEL
LIN {X 0,Y 288.239,Z 521.108,A -85,B 0,C 180,E1 -17027.84,E2 -17027.84} C_VEL
LIN {X 0,Y 290.321,Z 511.973,A -85,B 0,C 180,E1 -17029.811,E2 -17029.811} C_VEL
LIN {X 0,Y 292.533,Z 502.187,A -85,B 0,C 180,E1 -17031.493,E2 -17031.493} C_VEL
LIN {X 0,Y 294.781,Z 491.282,A -85,B 0,C 180,E1 -17032.98,E2 -17032.98} C_VEL
LIN {X 0,Y 296.946,Z 478.864,A -85,B 0,C 180,E1 -17034.282,E2 -17034.282} C_VEL
LIN {X 0,Y 298.692,Z 466.685,A -85,B 0,C 180,E1 -17035.244,E2 -17035.244} C_VEL
LIN {X 0,Y 300.109,Z 453.895,A -85,B 0,C 180,E1 -17035.953,E2 -17035.953} C_VEL
LIN {X 0,Y 300.954,Z 441.022,A -85,B 0,C 180,E1 -17036.415,E2 -17036.415} C_VEL
LIN {X 0,Y 302.77,Z 384.542,A -85,B 0,C 180,E1 -17037.759,E2 -17037.759} C_VEL
LIN {X 0,Y 299.425,Z 364.66,A -85,B 0,C 180,E1 -17038.704,E2 -17038.704} C_VEL
LIN {X 0,Y 296.629,Z 351.51,A -85,B 0,C 180,E1 -17039.418,E2 -17039.418} C_VEL
LIN {X 0,Y 290.903,Z 339.012,A -85,B 0,C 180,E1 -17040.52,E2 -17040.52} C_VEL
LIN {X 0,Y 289.477,Z 335.72,A -85,B 0,C 180,E1 -17040.831,E2 -17040.831} C_VEL
LIN {X 0,Y 286.938,Z 324.888,A -85,B 0,C 180,E1 -17044.69,E2 -17044.69} C_VEL
LIN {X 0,Y 284.324,Z 315.067,A -85,B 0,C 180,E1 -17048.506,E2 -17048.506} C_VEL
LIN {X 0,Y 284.271,Z 315.073,A -85,B 0,C 180,E1 -17052.124,E2 -17052.124} C_VEL
LIN {X 0,Y 284.257,Z 315.078,A -85,B 0,C 180,E1 -17056.189,E2 -17056.189} C_VEL
LIN {X 0,Y 284.308,Z 315.064,A -85,B 0,C 180,E1 -17060.024,E2 -17060.024} C_VEL
LIN {X 0,Y 284.332,Z 315.064,A -85,B 0,C 180,E1 -17063.614,E2 -17063.614} C_VEL
LIN {X 0,Y 284.309,Z 315.068,A -85,B 0,C 180,E1 -17067.189,E2 -17067.189} C_VEL
LIN {X 0,Y 284.36,Z 315.059,A -85,B 0,C 180,E1 -17070.376,E2 -17070.376} C_VEL
LIN {X 0,Y 284.379,Z 315.055,A -85,B 0,C 180,E1 -17073.586,E2 -17073.586} C_VEL
LIN {X 0,Y 284.367,Z 315.057,A -85,B 0,C 180,E1 -17076.707,E2 -17076.707} C_VEL
LIN {X 0,Y 284.404,Z 315.05,A -85,B 0,C 180,E1 -17081.261,E2 -17081.261} C_VEL
LIN {X 0,Y 284.493,Z 315.042,A -85,B 0,C 180,E1 -17084.459,E2 -17084.459} C_VEL
LIN {X 0,Y 284.488,Z 315.042,A -85,B 0,C 180,E1 -17088.601,E2 -17088.601} C_VEL
LIN {X 0,Y 284.64,Z 315.021,A -85,B 0,C 180,E1 -17091.48,E2 -17091.48} C_VEL
LIN {X 0,Y 284.597,Z 315.019,A -85,B 0,C 180,E1 -17094.331,E2 -17094.331} C_VEL
LIN {X 0,Y 284.854,Z 314.986,A -85,B 0,C 180,E1 -17098.586,E2 -17098.586} C_VEL
LIN {X 0,Y 284.854,Z 314.996,A -85,B 0,C 180,E1 -17101.414,E2 -17101.414} C_VEL
LIN {X 0,Y 284.698,Z 315.012,A -85,B 0,C 180,E1 -17107.09,E2 -17107.09} C_VEL
LIN {X 0,Y 284.567,Z 315.035,A -85,B 0,C 180,E1 -17109.955,E2 -17109.955} C_VEL
LIN {X 0,Y 284.482,Z 315.048,A -85,B 0,C 180,E1 -17114.303,E2 -17114.303} C_VEL
LIN {X 0,Y 284.425,Z 315.05,A -85,B 0,C 180,E1 -17117.248,E2 -17117.248} C_VEL
LIN {X 0,Y 284.378,Z 315.056,A -85,B 0,C 180,E1 -17120.242,E2 -17120.242} C_VEL
LIN {X 0,Y 284.337,Z 315.058,A -85,B 0,C 180,E1 -17124.846,E2 -17124.846} C_VEL
LIN {X 0,Y 284.328,Z 315.058,A -85,B 0,C 180,E1 -17128.011,E2 -17128.011} C_VEL
LIN {X 0,Y 284.294,Z 315.063,A -85,B 0,C 180,E1 -17131.274,E2 -17131.274} C_VEL
LIN {X 0,Y 284.341,Z 315.061,A -85,B 0,C 180,E1 -17135.348,E2 -17135.348} C_VEL
LIN {X 0,Y 284.312,Z 315.066,A -85,B 0,C 180,E1 -17138.169,E2 -17138.169} C_VEL
LIN {X 0,Y 284.27,Z 315.074,A -85,B 0,C 180,E1 -17142.124,E2 -17142.124} C_VEL
LIN {X 0,Y 284.256,Z 315.077,A -85,B 0,C 180,E1 -17146.189,E2 -17146.189} C_VEL
LIN {X 0,Y 284.302,Z 315.115,A -85,B 0,C 180,E1 -17147.344,E2 -17147.344} C_VEL
LIN {X 0,Y 285.218,Z 318.428,A -85,B 0,C 180,E1 -17148.631,E2 -17148.631} C_VEL
LIN {X 0,Y 294.429,Z 335.718,A -85,B 0,C 180,E1 -17150.403,E2 -17150.403} C_VEL
LIN {X 0,Y 300.493,Z 348.622,A -85,B 0,C 180,E1 -17151.533,E2 -17151.533} C_VEL
LIN {X 0,Y 303.69,Z 356.082,A -85,B 0,C 180,E1 -17152.123,E2 -17152.123} C_VEL
LIN {X 0,Y 301.201,Z 425.458,A -85,B 0,C 180,E1 -17153.773,E2 -17153.773} C_VEL
LIN {X 0,Y 300.14,Z 439.287,A -85,B 0,C 180,E1 -17154.376,E2 -17154.376} C_VEL
LIN {X 0,Y 299.016,Z 451.324,A -85,B 0,C 180,E1 -17155.181,E2 -17155.181} C_VEL
LIN {X 0,Y 297.323,Z 463.369,A -85,B 0,C 180,E1 -17156.256,E2 -17156.256} C_VEL
LIN {X 0,Y 295.392,Z 475.094,A -85,B 0,C 180,E1 -17157.634,E2 -17157.634} C_VEL
LIN {X 0,Y 293.339,Z 485.576,A -85,B 0,C 180,E1 -17159.195,E2 -17159.195} C_VEL
LIN {X 0,Y 291.027,Z 495.744,A -85,B 0,C 180,E1 -17161.119,E2 -17161.119} C_VEL
LIN {X 0,Y 288.865,Z 504.632,A -85,B 0,C 180,E1 -17163.25,E2 -17163.25} C_VEL
LIN {X 0,Y 287.088,Z 511.658,A -85,B 0,C 180,E1 -17165.407,E2 -17165.407} C_VEL
LIN {X 0,Y 285.596,Z 517.238,A -85,B 0,C 180,E1 -17167.577,E2 -17167.577} C_VEL
LIN {X 0,Y 284.374,Z 521.82,A -85,B 0,C 180,E1 -17169.906,E2 -17169.906} C_VEL
LIN {X 0,Y 283.828,Z 523.853,A -85,B 0,C 180,E1 -17171.222,E2 -17171.222} C_VEL
LIN {X 0,Y 283.303,Z 525.652,A -85,B 0,C 180,E1 -17172.681,E2 -17172.681} C_VEL
LIN {X 0,Y 282.951,Z 526.992,A -85,B 0,C 180,E1 -17174.143,E2 -17174.143} C_VEL
LIN {X 0,Y 282.66,Z 528.063,A -85,B 0,C 180,E1 -17175.856,E2 -17175.856} C_VEL
LIN {X 0,Y 282.325,Z 528.561,A -85,B 0,C 180,E1 -17178.512,E2 -17178.512} C_VEL
LIN {X 0,Y 282.3,Z 527.566,A -85,B 0,C 180,E1 -17181.409,E2 -17181.409} C_VEL
LIN {X 0,Y 282.423,Z 526.477,A -85,B 0,C 180,E1 -17182.852,E2 -17182.852} C_VEL
LIN {X 0,Y 282.61,Z 524.933,A -85,B 0,C 180,E1 -17184.291,E2 -17184.291} C_VEL
LIN {X 0,Y 282.794,Z 521.855,A -85,B 0,C 180,E1 -17186.437,E2 -17186.437} C_VEL
LIN {X 0,Y 283.281,Z 517.719,A -85,B 0,C 180,E1 -17188.578,E2 -17188.578} C_VEL
LIN {X 0,Y 283.966,Z 511.425,A -85,B 0,C 180,E1 -17191.063,E2 -17191.063} C_VEL
LIN {X 0,Y 285,Z 504.56,A -85,B 0,C 180,E1 -17193.18,E2 -17193.18} C_VEL
LIN {X 0,Y 286.181,Z 495.984,A -85,B 0,C 180,E1 -17195.283,E2 -17195.283} C_VEL
LIN {X 0,Y 287.386,Z 487.195,A -85,B 0,C 180,E1 -17197.023,E2 -17197.023} C_VEL
LIN {X 0,Y 288.826,Z 476.374,A -85,B 0,C 180,E1 -17198.747,E2 -17198.747} C_VEL
LIN {X 0,Y 290.181,Z 466.933,A -85,B 0,C 180,E1 -17199.936,E2 -17199.936} C_VEL
LIN {X 0,Y 291.403,Z 455.132,A -85,B 0,C 180,E1 -17201.124,E2 -17201.124} C_VEL
LIN {X 0,Y 292.244,Z 442.933,A -85,B 0,C 180,E1 -17202.058,E2 -17202.058} C_VEL
LIN {X 0,Y 292.861,Z 430.453,A -85,B 0,C 180,E1 -17202.736,E2 -17202.736} C_VEL
LIN {X 0,Y 293.578,Z 417.315,A -85,B 0,C 180,E1 -17203.144,E2 -17203.144} C_VEL
LIN {X 0,Y 295.195,Z 348.915,A -85,B 0,C 180,E1 -17204.782,E2 -17204.782} C_VEL
LIN {X 0,Y 293.765,Z 341.801,A -85,B 0,C 180,E1 -17205.075,E2 -17205.075} C_VEL
LIN {X 0,Y 287.871,Z 325.063,A -85,B 0,C 180,E1 -17205.983,E2 -17205.983} C_VEL
LIN {X 0,Y 284.959,Z 317.384,A -85,B 0,C 180,E1 -17206.457,E2 -17206.457} C_VEL
LIN {X 0,Y 284.447,Z 315.05,A -85,B 0,C 180,E1 -17207.339,E2 -17207.339} C_VEL
LIN {X 0,Y 284.365,Z 315.065,A -85,B 0,C 180,E1 -17210.242,E2 -17210.242} C_VEL
LIN {X 0,Y 284.319,Z 315.066,A -85,B 0,C 180,E1 -17213.852,E2 -17213.852} C_VEL
LIN {X 0,Y 284.279,Z 315.07,A -85,B 0,C 180,E1 -17218.015,E2 -17218.015} C_VEL
LIN {X 0,Y 284.281,Z 315.072,A -85,B 0,C 180,E1 -17221.275,E2 -17221.275} C_VEL
LIN {X 0,Y 284.333,Z 315.066,A -85,B 0,C 180,E1 -17225.346,E2 -17225.346} C_VEL
LIN {X 0,Y 284.296,Z 315.067,A -85,B 0,C 180,E1 -17228.17,E2 -17228.17} C_VEL
LIN {X 0,Y 284.232,Z 315.077,A -85,B 0,C 180,E1 -17232.116,E2 -17232.116} C_VEL
LIN {X 0,Y 284.25,Z 315.073,A -85,B 0,C 180,E1 -17236.188,E2 -17236.188} C_VEL
LIN {X 0,Y 284.301,Z 315.064,A -85,B 0,C 180,E1 -17240.023,E2 -17240.023} C_VEL
LIN {X 0,Y 284.323,Z 315.067,A -85,B 0,C 180,E1 -17243.613,E2 -17243.613} C_VEL
LIN {X 0,Y 284.302,Z 315.07,A -85,B 0,C 180,E1 -17247.189,E2 -17247.189} C_VEL
LIN {X 0,Y 284.352,Z 315.055,A -85,B 0,C 180,E1 -17250.375,E2 -17250.375} C_VEL
LIN {X 0,Y 284.371,Z 315.063,A -85,B 0,C 180,E1 -17253.586,E2 -17253.586} C_VEL
LIN {X 0,Y 284.323,Z 315.065,A -85,B 0,C 180,E1 -17254.83,E2 -17254.83} C_VEL
LIN {X 0,Y 283.681,Z 315.149,A -85,B 0,C 180,E1 -17256.012,E2 -17256.012} C_VEL
LIN {X 0,Y 280.864,Z 315.497,A -85,B 0,C 180,E1 -17257.937,E2 -17257.937} C_VEL
LIN {X 0,Y 278.455,Z 315.792,A -85,B 0,C 180,E1 -17259.501,E2 -17259.501} C_VEL
LIN {X 0,Y 277.411,Z 315.92,A -85,B 0,C 180,E1 -17260.712,E2 -17260.712} C_VEL
LIN {X 0,Y 277.321,Z 315.93,A -85,B 0,C 180,E1 -17261.123,E2 -17261.123} C_VEL
LIN {X 0,Y 277.428,Z 315.926,A -85,B 0,C 180,E1 -17265.326,E2 -17265.326} C_VEL
LIN {X 0,Y 277.453,Z 315.915,A -85,B 0,C 180,E1 -17269.787,E2 -17269.787} C_VEL
LIN {X 0,Y 277.604,Z 315.901,A -85,B 0,C 180,E1 -17272.728,E2 -17272.728} C_VEL
LIN {X 0,Y 277.813,Z 315.873,A -85,B 0,C 180,E1 -17278.551,E2 -17278.551} C_VEL
LIN {X 0,Y 277.814,Z 315.868,A -85,B 0,C 180,E1 -17281.45,E2 -17281.45} C_VEL
LIN {X 0,Y 277.642,Z 315.897,A -85,B 0,C 180,E1 -17287.271,E2 -17287.271} C_VEL
LIN {X 0,Y 277.5,Z 315.911,A -85,B 0,C 180,E1 -17290.212,E2 -17290.212} C_VEL
LIN {X 0,Y 277.422,Z 315.928,A -85,B 0,C 180,E1 -17294.675,E2 -17294.675} C_VEL
LIN {X 0,Y 277.339,Z 315.938,A -85,B 0,C 180,E1 -17299.234,E2 -17299.234} C_VEL
LIN {X 0,Y 277.314,Z 315.94,A -85,B 0,C 180,E1 -17304.171,E2 -17304.171} C_VEL
LIN {X 0,Y 277.321,Z 315.941,A -85,B 0,C 180,E1 -17307.506,E2 -17307.506} C_VEL
LIN {X 0,Y 277.267,Z 315.945,A -85,B 0,C 180,E1 -17310.482,E2 -17310.482} C_VEL
LIN {X 0,Y 277.25,Z 315.949,A -85,B 0,C 180,E1 -17313.896,E2 -17313.896} C_VEL
LIN {X 0,Y 277.277,Z 315.949,A -85,B 0,C 180,E1 -17317.468,E2 -17317.468} C_VEL
LIN {X 0,Y 277.206,Z 315.958,A -85,B 0,C 180,E1 -17321.238,E2 -17321.238} C_VEL
LIN {X 0,Y 277.197,Z 315.957,A -85,B 0,C 180,E1 -17325.228,E2 -17325.228} C_VEL
LIN {X 0,Y 277.22,Z 315.955,A -85,B 0,C 180,E1 -17329.513,E2 -17329.513} C_VEL
LIN {X 0,Y 277.269,Z 315.946,A -85,B 0,C 180,E1 -17332.533,E2 -17332.533} C_VEL
LIN {X 0,Y 277.279,Z 315.993,A -85,B 0,C 180,E1 -17336.654,E2 -17336.654} C_VEL
LIN {X 0,Y 279.931,Z 328.197,A -85,B 0,C 180,E1 -17340.687,E2 -17340.687} C_VEL
LIN {X 0,Y 281.459,Z 336.593,A -85,B 0,C 180,E1 -17343.292,E2 -17343.292} C_VEL
LIN {X 0,Y 283.825,Z 350.713,A -85,B 0,C 180,E1 -17343.871,E2 -17343.871} C_VEL
LIN {X 0,Y 287.865,Z 383.41,A -85,B 0,C 180,E1 -17345.06,E2 -17345.06} C_VEL
LIN {X 0,Y 286.3,Z 445.453,A -85,B 0,C 180,E1 -17346.614,E2 -17346.614} C_VEL
LIN {X 0,Y 285.419,Z 458.973,A -85,B 0,C 180,E1 -17347.23,E2 -17347.23} C_VEL
LIN {X 0,Y 284.381,Z 471.034,A -85,B 0,C 180,E1 -17348.052,E2 -17348.052} C_VEL
LIN {X 0,Y 283.112,Z 482.401,A -85,B 0,C 180,E1 -17349.094,E2 -17349.094} C_VEL
LIN {X 0,Y 281.499,Z 494.12,A -85,B 0,C 180,E1 -17350.494,E2 -17350.494} C_VEL
LIN {X 0,Y 280.131,Z 504.684,A -85,B 0,C 180,E1 -17352.103,E2 -17352.103} C_VEL
LIN {X 0,Y 278.881,Z 514.178,A -85,B 0,C 180,E1 -17353.907,E2 -17353.907} C_VEL
LIN {X 0,Y 277.514,Z 523.312,A -85,B 0,C 180,E1 -17356.08,E2 -17356.08} C_VEL
LIN {X 0,Y 276.444,Z 530.661,A -85,B 0,C 180,E1 -17358.266,E2 -17358.266} C_VEL
LIN {X 0,Y 275.861,Z 536.548,A -85,B 0,C 180,E1 -17360.469,E2 -17360.469} C_VEL
LIN {X 0,Y 275.485,Z 541.165,A -85,B 0,C 180,E1 -17362.672,E2 -17362.672} C_VEL
LIN {X 0,Y 275.336,Z 544.199,A -85,B 0,C 180,E1 -17364.555,E2 -17364.555} C_VEL
LIN {X 0,Y 275.327,Z 547.141,A -85,B 0,C 180,E1 -17367.074,E2 -17367.074} C_VEL
LIN {X 0,Y 275.313,Z 548.258,A -85,B 0,C 180,E1 -17368.538,E2 -17368.538} C_VEL
LIN {X 0,Y 275.331,Z 548.952,A -85,B 0,C 180,E1 -17370.001,E2 -17370.001} C_VEL
LIN {X 0,Y 275.29,Z 549.253,A -85,B 0,C 180,E1 -17371.464,E2 -17371.464} C_VEL
LIN {X 0,Y 275.284,Z 549.169,A -85,B 0,C 180,E1 -17372.928,E2 -17372.928} C_VEL
LIN {X 0,Y 275.286,Z 548.145,A -85,B 0,C 180,E1 -17375.335,E2 -17375.335} C_VEL
LIN {X 0,Y 275.49,Z 546.46,A -85,B 0,C 180,E1 -17377.329,E2 -17377.329} C_VEL
LIN {X 0,Y 275.963,Z 543.725,A -85,B 0,C 180,E1 -17379.529,E2 -17379.529} C_VEL
LIN {X 0,Y 276.774,Z 539.989,A -85,B 0,C 180,E1 -17381.721,E2 -17381.721} C_VEL
LIN {X 0,Y 277.917,Z 535.157,A -85,B 0,C 180,E1 -17383.901,E2 -17383.901} C_VEL
LIN {X 0,Y 279.907,Z 527.967,A -85,B 0,C 180,E1 -17386.408,E2 -17386.408} C_VEL
LIN {X 0,Y 281.747,Z 520.002,A -85,B 0,C 180,E1 -17388.578,E2 -17388.578} C_VEL
LIN {X 0,Y 284.097,Z 510.394,A -85,B 0,C 180,E1 -17390.642,E2 -17390.642} C_VEL
LIN {X 0,Y 286.452,Z 500.315,A -85,B 0,C 180,E1 -17392.352,E2 -17392.352} C_VEL
LIN {X 0,Y 288.796,Z 488.931,A -85,B 0,C 180,E1 -17393.865,E2 -17393.865} C_VEL
LIN {X 0,Y 290.814,Z 477.773,A -85,B 0,C 180,E1 -17395.019,E2 -17395.019} C_VEL
LIN {X 0,Y 292.667,Z 465.276,A -85,B 0,C 180,E1 -17395.993,E2 -17395.993} C_VEL
LIN {X 0,Y 294.118,Z 451.94,A -85,B 0,C 180,E1 -17396.714,E2 -17396.714} C_VEL
LIN {X 0,Y 294.947,Z 438.446,A -85,B 0,C 180,E1 -17397.173,E2 -17397.173} C_VEL
LIN {X 0,Y 296.638,Z 385.088,A -85,B 0,C 180,E1 -17398.468,E2 -17398.468} C_VEL
LIN {X 0,Y 292.972,Z 363.398,A -85,B 0,C 180,E1 -17399.541,E2 -17399.541} C_VEL
LIN {X 0,Y 290.954,Z 354.406,A -85,B 0,C 180,E1 -17400.063,E2 -17400.063} C_VEL
LIN {X 0,Y 284.208,Z 339.64,A -85,B 0,C 180,E1 -17401.422,E2 -17401.422} C_VEL
LIN {X 0,Y 282.349,Z 335.799,A -85,B 0,C 180,E1 -17401.806,E2 -17401.806} C_VEL
LIN {X 0,Y 282.054,Z 334.742,A -85,B 0,C 180,E1 -17402.093,E2 -17402.093} C_VEL
LIN {X 0,Y 279.544,Z 324.286,A -85,B 0,C 180,E1 -17405.999,E2 -17405.999} C_VEL
LIN {X 0,Y 277.268,Z 315.949,A -85,B 0,C 180,E1 -17409.432,E2 -17409.432} C_VEL
LIN {X 0,Y 277.211,Z 315.956,A -85,B 0,C 180,E1 -17413.198,E2 -17413.198} C_VEL
LIN {X 0,Y 277.217,Z 315.949,A -85,B 0,C 180,E1 -17417.325,E2 -17417.325} C_VEL
LIN {X 0,Y 277.263,Z 315.946,A -85,B 0,C 180,E1 -17421.793,E2 -17421.793} C_VEL
LIN {X 0,Y 277.285,Z 315.944,A -85,B 0,C 180,E1 -17424.341,E2 -17424.341} C_VEL
LIN {X 0,Y 277.246,Z 315.948,A -85,B 0,C 180,E1 -17427.836,E2 -17427.836} C_VEL
LIN {X 0,Y 277.291,Z 315.946,A -85,B 0,C 180,E1 -17431.212,E2 -17431.212} C_VEL
LIN {X 0,Y 277.315,Z 315.939,A -85,B 0,C 180,E1 -17434.479,E2 -17434.479} C_VEL
LIN {X 0,Y 277.286,Z 315.938,A -85,B 0,C 180,E1 -17437.655,E2 -17437.655} C_VEL
LIN {X 0,Y 277.346,Z 315.931,A -85,B 0,C 180,E1 -17440.766,E2 -17440.766} C_VEL
LIN {X 0,Y 277.435,Z 315.916,A -85,B 0,C 180,E1 -17445.326,E2 -17445.326} C_VEL
LIN {X 0,Y 277.462,Z 315.91,A -85,B 0,C 180,E1 -17449.787,E2 -17449.787} C_VEL
LIN {X 0,Y 277.641,Z 315.894,A -85,B 0,C 180,E1 -17452.729,E2 -17452.729} C_VEL
LIN {X 0,Y 277.82,Z 315.862,A -85,B 0,C 180,E1 -17458.55,E2 -17458.55} C_VEL
LIN {X 0,Y 277.82,Z 315.873,A -85,B 0,C 180,E1 -17461.449,E2 -17461.449} C_VEL
LIN {X 0,Y 277.653,Z 315.889,A -85,B 0,C 180,E1 -17467.271,E2 -17467.271} C_VEL
LIN {X 0,Y 277.507,Z 315.916,A -85,B 0,C 180,E1 -17470.211,E2 -17470.211} C_VEL
LIN {X 0,Y 277.435,Z 315.926,A -85,B 0,C 180,E1 -17474.674,E2 -17474.674} C_VEL
LIN {X 0,Y 277.345,Z 315.936,A -85,B 0,C 180,E1 -17479.234,E2 -17479.234} C_VEL
LIN {X 0,Y 277.292,Z 315.937,A -85,B 0,C 180,E1 -17484.157,E2 -17484.157} C_VEL
LIN {X 0,Y 277.324,Z 315.933,A -85,B 0,C 180,E1 -17487.504,E2 -17487.504} C_VEL
LIN {X 0,Y 277.272,Z 315.944,A -85,B 0,C 180,E1 -17490.481,E2 -17490.481} C_VEL
LIN {X 0,Y 277.247,Z 315.945,A -85,B 0,C 180,E1 -17493.896,E2 -17493.896} C_VEL
LIN {X 0,Y 277.268,Z 315.942,A -85,B 0,C 180,E1 -17497.469,E2 -17497.469} C_VEL
LIN {X 0,Y 277.21,Z 315.954,A -85,B 0,C 180,E1 -17501.236,E2 -17501.236} C_VEL
LIN {X 0,Y 277.202,Z 315.954,A -85,B 0,C 180,E1 -17505.226,E2 -17505.226} C_VEL
LIN {X 0,Y 277.234,Z 316.033,A -85,B 0,C 180,E1 -17506.472,E2 -17506.472} C_VEL
LIN {X 0,Y 277.96,Z 318.705,A -85,B 0,C 180,E1 -17507.56,E2 -17507.56} C_VEL
LIN {X 0,Y 287.104,Z 335.379,A -85,B 0,C 180,E1 -17509.41,E2 -17509.41} C_VEL
LIN {X 0,Y 293.918,Z 349.365,A -85,B 0,C 180,E1 -17510.731,E2 -17510.731} C_VEL
LIN {X 0,Y 297.552,Z 357.947,A -85,B 0,C 180,E1 -17511.434,E2 -17511.434} C_VEL
LIN {X 0,Y 295.052,Z 426.224,A -85,B 0,C 180,E1 -17513.1,E2 -17513.1} C_VEL
LIN {X 0,Y 293.948,Z 439.98,A -85,B 0,C 180,E1 -17513.719,E2 -17513.719} C_VEL
LIN {X 0,Y 292.697,Z 452.644,A -85,B 0,C 180,E1 -17514.6,E2 -17514.6} C_VEL
LIN {X 0,Y 290.933,Z 464.312,A -85,B 0,C 180,E1 -17515.68,E2 -17515.68} C_VEL
LIN {X 0,Y 289.001,Z 475.53,A -85,B 0,C 180,E1 -17517.035,E2 -17517.035} C_VEL
LIN {X 0,Y 286.864,Z 485.97,A -85,B 0,C 180,E1 -17518.626,E2 -17518.626} C_VEL
LIN {X 0,Y 284.662,Z 495.28,A -85,B 0,C 180,E1 -17520.41,E2 -17520.41} C_VEL
LIN {X 0,Y 282.338,Z 504.302,A -85,B 0,C 180,E1 -17522.58,E2 -17522.58} C_VEL
LIN {X 0,Y 280.418,Z 511.472,A -85,B 0,C 180,E1 -17524.782,E2 -17524.782} C_VEL
LIN {X 0,Y 278.847,Z 517.144,A -85,B 0,C 180,E1 -17527.004,E2 -17527.004} C_VEL
LIN {X 0,Y 277.443,Z 522.158,A -85,B 0,C 180,E1 -17529.596,E2 -17529.596} C_VEL
LIN {X 0,Y 276.349,Z 525.753,A -85,B 0,C 180,E1 -17532.23,E2 -17532.23} C_VEL
LIN {X 0,Y 275.957,Z 527.136,A -85,B 0,C 180,E1 -17533.731,E2 -17533.731} C_VEL
LIN {X 0,Y 275.588,Z 528.358,A -85,B 0,C 180,E1 -17535.712,E2 -17535.712} C_VEL
LIN {X 0,Y 275.251,Z 528.847,A -85,B 0,C 180,E1 -17538.213,E2 -17538.213} C_VEL
LIN {X 0,Y 275.209,Z 527.921,A -85,B 0,C 180,E1 -17541.186,E2 -17541.186} C_VEL
LIN {X 0,Y 275.299,Z 526.876,A -85,B 0,C 180,E1 -17542.666,E2 -17542.666} C_VEL
LIN {X 0,Y 275.502,Z 525.326,A -85,B 0,C 180,E1 -17544.199,E2 -17544.199} C_VEL
LIN {X 0,Y 275.709,Z 522.391,A -85,B 0,C 180,E1 -17546.346,E2 -17546.346} C_VEL
LIN {X 0,Y 276.17,Z 518.338,A -85,B 0,C 180,E1 -17548.541,E2 -17548.541} C_VEL
LIN {X 0,Y 276.879,Z 512.129,A -85,B 0,C 180,E1 -17551.09,E2 -17551.09} C_VEL
LIN {X 0,Y 277.913,Z 505.363,A -85,B 0,C 180,E1 -17553.261,E2 -17553.261} C_VEL
LIN {X 0,Y 279.15,Z 496.956,A -85,B 0,C 180,E1 -17555.417,E2 -17555.417} C_VEL
LIN {X 0,Y 280.376,Z 488.309,A -85,B 0,C 180,E1 -17557.199,E2 -17557.199} C_VEL
LIN {X 0,Y 281.853,Z 477.663,A -85,B 0,C 180,E1 -17558.965,E2 -17558.965} C_VEL
LIN {X 0,Y 283.405,Z 467.017,A -85,B 0,C 180,E1 -17560.357,E2 -17560.357} C_VEL
LIN {X 0,Y 284.68,Z 455.15,A -85,B 0,C 180,E1 -17561.57,E2 -17561.57} C_VEL
LIN {X 0,Y 285.55,Z 442.88,A -85,B 0,C 180,E1 -17562.526,E2 -17562.526} C_VEL
LIN {X 0,Y 286.141,Z 431.182,A -85,B 0,C 180,E1 -17563.176,E2 -17563.176} C_VEL
LIN {X 0,Y 286.86,Z 418.501,A -85,B 0,C 180,E1 -17563.593,E2 -17563.593} C_VEL
LIN {X 0,Y 288.565,Z 349.689,A -85,B 0,C 180,E1 -17565.275,E2 -17565.275} C_VEL
LIN {X 0,Y 287.405,Z 344.038,A -85,B 0,C 180,E1 -17565.517,E2 -17565.517} C_VEL
LIN {X 0,Y 281.727,Z 327.895,A -85,B 0,C 180,E1 -17566.423,E2 -17566.423} C_VEL
LIN {X 0,Y 277.747,Z 317.601,A -85,B 0,C 180,E1 -17567.099,E2 -17567.099} C_VEL
LIN {X 0,Y 277.384,Z 315.932,A -85,B 0,C 180,E1 -17567.699,E2 -17567.699} C_VEL
LIN {X 0,Y 277.281,Z 315.946,A -85,B 0,C 180,E1 -17570.783,E2 -17570.783} C_VEL
LIN {X 0,Y 277.275,Z 315.945,A -85,B 0,C 180,E1 -17574.15,E2 -17574.15} C_VEL
LIN {X 0,Y 277.266,Z 315.943,A -85,B 0,C 180,E1 -17577.481,E2 -17577.481} C_VEL
LIN {X 0,Y 277.245,Z 315.949,A -85,B 0,C 180,E1 -17580.472,E2 -17580.472} C_VEL
LIN {X 0,Y 277.242,Z 315.948,A -85,B 0,C 180,E1 -17583.895,E2 -17583.895} C_VEL
LIN {X 0,Y 277.256,Z 315.945,A -85,B 0,C 180,E1 -17587.47,E2 -17587.47} C_VEL
LIN {X 0,Y 277.179,Z 315.958,A -85,B 0,C 180,E1 -17591.24,E2 -17591.24} C_VEL
LIN {X 0,Y 277.193,Z 315.953,A -85,B 0,C 180,E1 -17595.226,E2 -17595.226} C_VEL
LIN {X 0,Y 277.217,Z 315.949,A -85,B 0,C 180,E1 -17599.511,E2 -17599.511} C_VEL
LIN {X 0,Y 277.256,Z 315.94,A -85,B 0,C 180,E1 -17602.529,E2 -17602.529} C_VEL
LIN {X 0,Y 277.241,Z 315.947,A -85,B 0,C 180,E1 -17606.104,E2 -17606.104} C_VEL
LIN {X 0,Y 277.255,Z 315.94,A -85,B 0,C 180,E1 -17609.538,E2 -17609.538} C_VEL
LIN {X 0,Y 277.353,Z 315.932,A -85,B 0,C 180,E1 -17612.864,E2 -17612.864} C_VEL
LIN {X 0,Y 277.291,Z 315.942,A -85,B 0,C 180,E1 -17616.076,E2 -17616.076} C_VEL
LIN {X 0,Y 277.335,Z 315.929,A -85,B 0,C 180,E1 -17620.766,E2 -17620.766} C_VEL
LIN {X 0,Y 277.321,Z 315.93,A -85,B 0,C 180,E1 -17621.123,E2 -17621.123} C_VEL
LIN {X 0,Y 276.639,Z 316.023,A -85,B 0,C 180,E1 -17622.336,E2 -17622.336} C_VEL
LIN {X 0,Y 273.787,Z 316.38,A -85,B 0,C 180,E1 -17624.313,E2 -17624.313} C_VEL
LIN {X 0,Y 271.404,Z 316.679,A -85,B 0,C 180,E1 -17625.92,E2 -17625.92} C_VEL
LIN {X 0,Y 270.421,Z 316.796,A -85,B 0,C 180,E1 -17627.165,E2 -17627.165} C_VEL
LIN {X 0,Y 270.361,Z 316.8,A -85,B 0,C 180,E1 -17627.586,E2 -17627.586} C_VEL
LIN {X 0,Y 270.52,Z 316.777,A -85,B 0,C 180,E1 -17631.032,E2 -17631.032} C_VEL
LIN {X 0,Y 270.514,Z 316.788,A -85,B 0,C 180,E1 -17634.035,E2 -17634.035} C_VEL
LIN {X 0,Y 270.779,Z 316.749,A -85,B 0,C 180,E1 -17638.513,E2 -17638.513} C_VEL
LIN {X 0,Y 270.78,Z 316.743,A -85,B 0,C 180,E1 -17641.487,E2 -17641.487} C_VEL
LIN {X 0,Y 270.601,Z 316.774,A -85,B 0,C 180,E1 -17647.462,E2 -17647.462} C_VEL
LIN {X 0,Y 270.435,Z 316.789,A -85,B 0,C 180,E1 -17650.481,E2 -17650.481} C_VEL
LIN {X 0,Y 270.39,Z 316.804,A -85,B 0,C 180,E1 -17655.066,E2 -17655.066} C_VEL
LIN {X 0,Y 270.296,Z 316.813,A -85,B 0,C 180,E1 -17659.756,E2 -17659.756} C_VEL
LIN {X 0,Y 270.269,Z 316.819,A -85,B 0,C 180,E1 -17664.586,E2 -17664.586} C_VEL
LIN {X 0,Y 270.267,Z 316.818,A -85,B 0,C 180,E1 -17667.909,E2 -17667.909} C_VEL
LIN {X 0,Y 270.18,Z 316.833,A -85,B 0,C 180,E1 -17671.349,E2 -17671.349} C_VEL
LIN {X 0,Y 270.21,Z 316.827,A -85,B 0,C 180,E1 -17674.905,E2 -17674.905} C_VEL
LIN {X 0,Y 270.218,Z 316.826,A -85,B 0,C 180,E1 -17678.718,E2 -17678.718} C_VEL
LIN {X 0,Y 270.161,Z 316.835,A -85,B 0,C 180,E1 -17683.25,E2 -17683.25} C_VEL
LIN {X 0,Y 270.169,Z 316.834,A -85,B 0,C 180,E1 -17687.443,E2 -17687.443} C_VEL
LIN {X 0,Y 270.205,Z 316.828,A -85,B 0,C 180,E1 -17691.375,E2 -17691.375} C_VEL
LIN {X 0,Y 270.203,Z 316.829,A -85,B 0,C 180,E1 -17695.096,E2 -17695.096} C_VEL
LIN {X 0,Y 270.237,Z 316.955,A -85,B 0,C 180,E1 -17696.218,E2 -17696.218} C_VEL
LIN {X 0,Y 272.879,Z 328.875,A -85,B 0,C 180,E1 -17700.28,E2 -17700.28} C_VEL
LIN {X 0,Y 274.274,Z 336.351,A -85,B 0,C 180,E1 -17702.658,E2 -17702.658} C_VEL
LIN {X 0,Y 275.758,Z 341.505,A -85,B 0,C 180,E1 -17702.934,E2 -17702.934} C_VEL
LIN {X 0,Y 279.838,Z 371.778,A -85,B 0,C 180,E1 -17704.114,E2 -17704.114} C_VEL
LIN {X 0,Y 281.247,Z 383.938,A -85,B 0,C 180,E1 -17704.558,E2 -17704.558} C_VEL
LIN {X 0,Y 279.624,Z 445.246,A -85,B 0,C 180,E1 -17706.127,E2 -17706.127} C_VEL
LIN {X 0,Y 278.727,Z 458.632,A -85,B 0,C 180,E1 -17706.75,E2 -17706.75} C_VEL
LIN {X 0,Y 277.671,Z 470.716,A -85,B 0,C 180,E1 -17707.591,E2 -17707.591} C_VEL
LIN {X 0,Y 276.247,Z 482.897,A -85,B 0,C 180,E1 -17708.745,E2 -17708.745} C_VEL
LIN {X 0,Y 274.586,Z 494.476,A -85,B 0,C 180,E1 -17710.177,E2 -17710.177} C_VEL
LIN {X 0,Y 273.177,Z 504.933,A -85,B 0,C 180,E1 -17711.825,E2 -17711.825} C_VEL
LIN {X 0,Y 271.993,Z 513.468,A -85,B 0,C 180,E1 -17713.488,E2 -17713.488} C_VEL
LIN {X 0,Y 270.6,Z 522.69,A -85,B 0,C 180,E1 -17715.717,E2 -17715.717} C_VEL
LIN {X 0,Y 269.448,Z 530.1,A -85,B 0,C 180,E1 -17717.957,E2 -17717.957} C_VEL
LIN {X 0,Y 268.807,Z 536.046,A -85,B 0,C 180,E1 -17720.216,E2 -17720.216} C_VEL
LIN {X 0,Y 268.403,Z 540.719,A -85,B 0,C 180,E1 -17722.478,E2 -17722.478} C_VEL
LIN {X 0,Y 268.232,Z 544.141,A -85,B 0,C 180,E1 -17724.654,E2 -17724.654} C_VEL
LIN {X 0,Y 268.234,Z 546.781,A -85,B 0,C 180,E1 -17726.997,E2 -17726.997} C_VEL
LIN {X 0,Y 268.238,Z 547.94,A -85,B 0,C 180,E1 -17728.499,E2 -17728.499} C_VEL
LIN {X 0,Y 268.252,Z 548.656,A -85,B 0,C 180,E1 -17730.001,E2 -17730.001} C_VEL
LIN {X 0,Y 268.215,Z 548.979,A -85,B 0,C 180,E1 -17731.502,E2 -17731.502} C_VEL
LIN {X 0,Y 268.194,Z 548.914,A -85,B 0,C 180,E1 -17733.005,E2 -17733.005} C_VEL
LIN {X 0,Y 268.179,Z 548.07,A -85,B 0,C 180,E1 -17735.224,E2 -17735.224} C_VEL
LIN {X 0,Y 268.414,Z 546.289,A -85,B 0,C 180,E1 -17737.523,E2 -17737.523} C_VEL
LIN {X 0,Y 268.951,Z 543.598,A -85,B 0,C 180,E1 -17739.78,E2 -17739.78} C_VEL
LIN {X 0,Y 269.777,Z 539.909,A -85,B 0,C 180,E1 -17742.03,E2 -17742.03} C_VEL
LIN {X 0,Y 271.019,Z 535.128,A -85,B 0,C 180,E1 -17744.262,E2 -17744.262} C_VEL
LIN {X 0,Y 273.071,Z 527.998,A -85,B 0,C 180,E1 -17746.831,E2 -17746.831} C_VEL
LIN {X 0,Y 274.893,Z 520.652,A -85,B 0,C 180,E1 -17748.922,E2 -17748.922} C_VEL
LIN {X 0,Y 277.026,Z 512.385,A -85,B 0,C 180,E1 -17750.805,E2 -17750.805} C_VEL
LIN {X 0,Y 279.409,Z 502.792,A -85,B 0,C 180,E1 -17752.556,E2 -17752.556} C_VEL
LIN {X 0,Y 281.804,Z 492.166,A -85,B 0,C 180,E1 -17754.104,E2 -17754.104} C_VEL
LIN {X 0,Y 283.875,Z 481.902,A -85,B 0,C 180,E1 -17755.282,E2 -17755.282} C_VEL
LIN {X 0,Y 285.826,Z 469.693,A -85,B 0,C 180,E1 -17756.368,E2 -17756.368} C_VEL
LIN {X 0,Y 287.594,Z 456.111,A -85,B 0,C 180,E1 -17757.222,E2 -17757.222} C_VEL
LIN {X 0,Y 288.65,Z 443.535,A -85,B 0,C 180,E1 -17757.745,E2 -17757.745} C_VEL
LIN {X 0,Y 290.627,Z 386.2,A -85,B 0,C 180,E1 -17759.181,E2 -17759.181} C_VEL
LIN {X 0,Y 286.835,Z 363.798,A -85,B 0,C 180,E1 -17760.333,E2 -17760.333} C_VEL
LIN {X 0,Y 285.427,Z 357.507,A -85,B 0,C 180,E1 -17760.712,E2 -17760.712} C_VEL
LIN {X 0,Y 279.064,Z 343.58,A -85,B 0,C 180,E1 -17762.046,E2 -17762.046} C_VEL
LIN {X 0,Y 274.845,Z 334.952,A -85,B 0,C 180,E1 -17763.007,E2 -17763.007} C_VEL
LIN {X 0,Y 272.821,Z 326.335,A -85,B 0,C 180,E1 -17766.334,E2 -17766.334} C_VEL
LIN {X 0,Y 270.199,Z 316.826,A -85,B 0,C 180,E1 -17770.353,E2 -17770.353} C_VEL
LIN {X 0,Y 270.154,Z 316.831,A -85,B 0,C 180,E1 -17774.62,E2 -17774.62} C_VEL
LIN {X 0,Y 270.171,Z 316.829,A -85,B 0,C 180,E1 -17778.972,E2 -17778.972} C_VEL
LIN {X 0,Y 270.217,Z 316.82,A -85,B 0,C 180,E1 -17783.259,E2 -17783.259} C_VEL
LIN {X 0,Y 270.204,Z 316.821,A -85,B 0,C 180,E1 -17786.892,E2 -17786.892} C_VEL
LIN {X 0,Y 270.23,Z 316.819,A -85,B 0,C 180,E1 -17790.387,E2 -17790.387} C_VEL
LIN {X 0,Y 270.265,Z 316.813,A -85,B 0,C 180,E1 -17793.764,E2 -17793.764} C_VEL
LIN {X 0,Y 270.234,Z 316.816,A -85,B 0,C 180,E1 -17797.039,E2 -17797.039} C_VEL
LIN {X 0,Y 270.303,Z 316.811,A -85,B 0,C 180,E1 -17800.244,E2 -17800.244} C_VEL
LIN {X 0,Y 270.404,Z 316.794,A -85,B 0,C 180,E1 -17804.935,E2 -17804.935} C_VEL
LIN {X 0,Y 270.414,Z 316.789,A -85,B 0,C 180,E1 -17809.518,E2 -17809.518} C_VEL
LIN {X 0,Y 270.599,Z 316.771,A -85,B 0,C 180,E1 -17812.538,E2 -17812.538} C_VEL
LIN {X 0,Y 270.786,Z 316.738,A -85,B 0,C 180,E1 -17818.513,E2 -17818.513} C_VEL
LIN {X 0,Y 270.786,Z 316.749,A -85,B 0,C 180,E1 -17821.487,E2 -17821.487} C_VEL
LIN {X 0,Y 270.611,Z 316.765,A -85,B 0,C 180,E1 -17827.461,E2 -17827.461} C_VEL
LIN {X 0,Y 270.442,Z 316.795,A -85,B 0,C 180,E1 -17830.481,E2 -17830.481} C_VEL
LIN {X 0,Y 270.403,Z 316.8,A -85,B 0,C 180,E1 -17835.064,E2 -17835.064} C_VEL
LIN {X 0,Y 270.302,Z 316.812,A -85,B 0,C 180,E1 -17839.755,E2 -17839.755} C_VEL
LIN {X 0,Y 270.238,Z 316.814,A -85,B 0,C 180,E1 -17844.589,E2 -17844.589} C_VEL
LIN {X 0,Y 270.27,Z 316.809,A -85,B 0,C 180,E1 -17847.909,E2 -17847.909} C_VEL
LIN {X 0,Y 270.184,Z 316.82,A -85,B 0,C 180,E1 -17851.348,E2 -17851.348} C_VEL
LIN {X 0,Y 270.202,Z 316.82,A -85,B 0,C 180,E1 -17854.905,E2 -17854.905} C_VEL
LIN {X 0,Y 270.198,Z 316.827,A -85,B 0,C 180,E1 -17858.71,E2 -17858.71} C_VEL
LIN {X 0,Y 270.166,Z 316.831,A -85,B 0,C 180,E1 -17863.249,E2 -17863.249} C_VEL
LIN {X 0,Y 270.167,Z 316.86,A -85,B 0,C 180,E1 -17865.504,E2 -17865.504} C_VEL
LIN {X 0,Y 270.777,Z 318.982,A -85,B 0,C 180,E1 -17866.426,E2 -17866.426} C_VEL
LIN {X 0,Y 272.935,Z 322.822,A -85,B 0,C 180,E1 -17866.903,E2 -17866.903} C_VEL
LIN {X 0,Y 281.778,Z 338.853,A -85,B 0,C 180,E1 -17868.759,E2 -17868.759} C_VEL
LIN {X 0,Y 288.621,Z 353.025,A -85,B 0,C 180,E1 -17870.142,E2 -17870.142} C_VEL
LIN {X 0,Y 291.586,Z 360.134,A -85,B 0,C 180,E1 -17870.741,E2 -17870.741} C_VEL
LIN {X 0,Y 289.024,Z 426.013,A -85,B 0,C 180,E1 -17872.365,E2 -17872.365} C_VEL
LIN {X 0,Y 287.981,Z 439.132,A -85,B 0,C 180,E1 -17872.952,E2 -17872.952} C_VEL
LIN {X 0,Y 286.812,Z 449.793,A -85,B 0,C 180,E1 -17873.652,E2 -17873.652} C_VEL
LIN {X 0,Y 285.115,Z 462.443,A -85,B 0,C 180,E1 -17874.782,E2 -17874.782} C_VEL
LIN {X 0,Y 283.19,Z 473.339,A -85,B 0,C 180,E1 -17876.055,E2 -17876.055} C_VEL
LIN {X 0,Y 280.902,Z 484.229,A -85,B 0,C 180,E1 -17877.67,E2 -17877.67} C_VEL
LIN {X 0,Y 278.729,Z 493.221,A -85,B 0,C 180,E1 -17879.331,E2 -17879.331} C_VEL
LIN {X 0,Y 276.646,Z 501.168,A -85,B 0,C 180,E1 -17881.139,E2 -17881.139} C_VEL
LIN {X 0,Y 274.463,Z 508.931,A -85,B 0,C 180,E1 -17883.346,E2 -17883.346} C_VEL
LIN {X 0,Y 272.661,Z 515.259,A -85,B 0,C 180,E1 -17885.643,E2 -17885.643} C_VEL
LIN {X 0,Y 271.178,Z 520.172,A -85,B 0,C 180,E1 -17887.926,E2 -17887.926} C_VEL
LIN {X 0,Y 270.024,Z 523.913,A -85,B 0,C 180,E1 -17890.223,E2 -17890.223} C_VEL
LIN {X 0,Y 269.406,Z 525.829,A -85,B 0,C 180,E1 -17891.757,E2 -17891.757} C_VEL
LIN {X 0,Y 268.968,Z 527.279,A -85,B 0,C 180,E1 -17893.296,E2 -17893.296} C_VEL
LIN {X 0,Y 268.544,Z 528.64,A -85,B 0,C 180,E1 -17895.538,E2 -17895.538} C_VEL
LIN {X 0,Y 268.195,Z 529.118,A -85,B 0,C 180,E1 -17897.898,E2 -17897.898} C_VEL
LIN {X 0,Y 268.056,Z 528.901,A -85,B 0,C 180,E1 -17899.424,E2 -17899.424} C_VEL
LIN {X 0,Y 268.102,Z 528.277,A -85,B 0,C 180,E1 -17900.95,E2 -17900.95} C_VEL
LIN {X 0,Y 268.206,Z 527.266,A -85,B 0,C 180,E1 -17902.471,E2 -17902.471} C_VEL
LIN {X 0,Y 268.418,Z 525.554,A -85,B 0,C 180,E1 -17904.242,E2 -17904.242} C_VEL
LIN {X 0,Y 268.682,Z 521.688,A -85,B 0,C 180,E1 -17907,E2 -17907} C_VEL
LIN {X 0,Y 269.256,Z 517.343,A -85,B 0,C 180,E1 -17909.251,E2 -17909.251} C_VEL
LIN {X 0,Y 269.941,Z 511.828,A -85,B 0,C 180,E1 -17911.491,E2 -17911.491} C_VEL
LIN {X 0,Y 271.056,Z 504.933,A -85,B 0,C 180,E1 -17913.716,E2 -17913.716} C_VEL
LIN {X 0,Y 272.34,Z 496.311,A -85,B 0,C 180,E1 -17915.924,E2 -17915.924} C_VEL
LIN {X 0,Y 273.661,Z 487.481,A -85,B 0,C 180,E1 -17917.748,E2 -17917.748} C_VEL
LIN {X 0,Y 275.049,Z 477.781,A -85,B 0,C 180,E1 -17919.374,E2 -17919.374} C_VEL
LIN {X 0,Y 276.647,Z 467.096,A -85,B 0,C 180,E1 -17920.798,E2 -17920.798} C_VEL
LIN {X 0,Y 277.813,Z 457.116,A -85,B 0,C 180,E1 -17921.86,E2 -17921.86} C_VEL
LIN {X 0,Y 278.703,Z 445.391,A -85,B 0,C 180,E1 -17922.839,E2 -17922.839} C_VEL
LIN {X 0,Y 279.375,Z 432.807,A -85,B 0,C 180,E1 -17923.594,E2 -17923.594} C_VEL
LIN {X 0,Y 280.188,Z 419.594,A -85,B 0,C 180,E1 -17924.062,E2 -17924.062} C_VEL
LIN {X 0,Y 281.948,Z 350.411,A -85,B 0,C 180,E1 -17925.792,E2 -17925.792} C_VEL
LIN {X 0,Y 280.752,Z 345.086,A -85,B 0,C 180,E1 -17926.037,E2 -17926.037} C_VEL
LIN {X 0,Y 273.731,Z 325.885,A -85,B 0,C 180,E1 -17927.185,E2 -17927.185} C_VEL
LIN {X 0,Y 270.59,Z 317.965,A -85,B 0,C 180,E1 -17927.72,E2 -17927.72} C_VEL
LIN {X 0,Y 270.319,Z 316.813,A -85,B 0,C 180,E1 -17928.178,E2 -17928.178} C_VEL
LIN {X 0,Y 270.204,Z 316.826,A -85,B 0,C 180,E1 -17931.353,E2 -17931.353} C_VEL
LIN {X 0,Y 270.221,Z 316.825,A -85,B 0,C 180,E1 -17934.589,E2 -17934.589} C_VEL
LIN {X 0,Y 270.195,Z 316.824,A -85,B 0,C 180,E1 -17937.916,E2 -17937.916} C_VEL
LIN {X 0,Y 270.17,Z 316.829,A -85,B 0,C 180,E1 -17941.349,E2 -17941.349} C_VEL
LIN {X 0,Y 270.195,Z 316.829,A -85,B 0,C 180,E1 -17944.905,E2 -17944.905} C_VEL
LIN {X 0,Y 270.194,Z 316.825,A -85,B 0,C 180,E1 -17948.709,E2 -17948.709} C_VEL
LIN {X 0,Y 270.143,Z 316.829,A -85,B 0,C 180,E1 -17953.244,E2 -17953.244} C_VEL
LIN {X 0,Y 270.166,Z 316.831,A -85,B 0,C 180,E1 -17957.441,E2 -17957.441} C_VEL
LIN {X 0,Y 270.202,Z 316.819,A -85,B 0,C 180,E1 -17961.373,E2 -17961.373} C_VEL
LIN {X 0,Y 270.195,Z 316.827,A -85,B 0,C 180,E1 -17965.094,E2 -17965.094} C_VEL
LIN {X 0,Y 270.194,Z 316.821,A -85,B 0,C 180,E1 -17969.13,E2 -17969.13} C_VEL
LIN {X 0,Y 270.258,Z 316.817,A -85,B 0,C 180,E1 -17972.145,E2 -17972.145} C_VEL
LIN {X 0,Y 270.232,Z 316.825,A -85,B 0,C 180,E1 -17975.537,E2 -17975.537} C_VEL
LIN {X 0,Y 270.293,Z 316.807,A -85,B 0,C 180,E1 -17980.244,E2 -17980.244} C_VEL
LIN {X 0,Y 270.396,Z 316.801,A -85,B 0,C 180,E1 -17984.935,E2 -17984.935} C_VEL
LIN {X 0,Y 270.361,Z 316.8,A -85,B 0,C 180,E1 -17987.586,E2 -17987.586} C_VEL
LIN {X 0,Y 269.779,Z 316.876,A -85,B 0,C 180,E1 -17988.83,E2 -17988.83} C_VEL
LIN {X 0,Y 267.055,Z 317.22,A -85,B 0,C 180,E1 -17990.861,E2 -17990.861} C_VEL
LIN {X 0,Y 263.824,Z 317.621,A -85,B 0,C 180,E1 -17993.358,E2 -17993.358} C_VEL
LIN {X 0,Y 263.441,Z 317.665,A -85,B 0,C 180,E1 -17994.221,E2 -17994.221} C_VEL
LIN {X 0,Y 263.743,Z 317.625,A -85,B 0,C 180,E1 -17998.473,E2 -17998.473} C_VEL
LIN {X 0,Y 263.744,Z 317.619,A -85,B 0,C 180,E1 -18001.527,E2 -18001.527} C_VEL
LIN {X 0,Y 263.563,Z 317.651,A -85,B 0,C 180,E1 -18007.662,E2 -18007.662} C_VEL
LIN {X 0,Y 263.367,Z 317.667,A -85,B 0,C 180,E1 -18010.766,E2 -18010.766} C_VEL
LIN {X 0,Y 263.339,Z 317.68,A -85,B 0,C 180,E1 -18015.479,E2 -18015.479} C_VEL
LIN {X 0,Y 263.258,Z 317.691,A -85,B 0,C 180,E1 -18020.307,E2 -18020.307} C_VEL
LIN {X 0,Y 263.203,Z 317.698,A -85,B 0,C 180,E1 -18025.292,E2 -18025.292} C_VEL
LIN {X 0,Y 263.175,Z 317.704,A -85,B 0,C 180,E1 -18028.73,E2 -18028.73} C_VEL
LIN {X 0,Y 263.129,Z 317.708,A -85,B 0,C 180,E1 -18032.289,E2 -18032.289} C_VEL
LIN {X 0,Y 263.183,Z 317.701,A -85,B 0,C 180,E1 -18035.979,E2 -18035.979} C_VEL
LIN {X 0,Y 263.111,Z 317.711,A -85,B 0,C 180,E1 -18039.872,E2 -18039.872} C_VEL
LIN {X 0,Y 263.1,Z 317.713,A -85,B 0,C 180,E1 -18043.989,E2 -18043.989} C_VEL
LIN {X 0,Y 263.121,Z 317.708,A -85,B 0,C 180,E1 -18048.408,E2 -18048.408} C_VEL
LIN {X 0,Y 263.182,Z 317.702,A -85,B 0,C 180,E1 -18053.237,E2 -18053.237} C_VEL
LIN {X 0,Y 263.174,Z 317.856,A -85,B 0,C 180,E1 -18055.735,E2 -18055.735} C_VEL
LIN {X 0,Y 265.732,Z 329.524,A -85,B 0,C 180,E1 -18059.835,E2 -18059.835} C_VEL
LIN {X 0,Y 267.015,Z 336.031,A -85,B 0,C 180,E1 -18061.98,E2 -18061.98} C_VEL
LIN {X 0,Y 269.318,Z 342.986,A -85,B 0,C 180,E1 -18062.396,E2 -18062.396} C_VEL
LIN {X 0,Y 273.366,Z 373.671,A -85,B 0,C 180,E1 -18063.624,E2 -18063.624} C_VEL
LIN {X 0,Y 274.637,Z 384.349,A -85,B 0,C 180,E1 -18064.029,E2 -18064.029} C_VEL
LIN {X 0,Y 272.991,Z 444.588,A -85,B 0,C 180,E1 -18065.602,E2 -18065.602} C_VEL
LIN {X 0,Y 272.063,Z 458.247,A -85,B 0,C 180,E1 -18066.247,E2 -18066.247} C_VEL
LIN {X 0,Y 270.959,Z 470.363,A -85,B 0,C 180,E1 -18067.105,E2 -18067.105} C_VEL
LIN {X 0,Y 269.603,Z 481.774,A -85,B 0,C 180,E1 -18068.195,E2 -18068.195} C_VEL
LIN {X 0,Y 267.901,Z 493.517,A -85,B 0,C 180,E1 -18069.661,E2 -18069.661} C_VEL
LIN {X 0,Y 266.367,Z 504.09,A -85,B 0,C 180,E1 -18071.343,E2 -18071.343} C_VEL
LIN {X 0,Y 265.103,Z 512.728,A -85,B 0,C 180,E1 -18073.046,E2 -18073.046} C_VEL
LIN {X 0,Y 263.878,Z 520.675,A -85,B 0,C 180,E1 -18074.95,E2 -18074.95} C_VEL
LIN {X 0,Y 262.665,Z 528.412,A -85,B 0,C 180,E1 -18077.248,E2 -18077.248} C_VEL
LIN {X 0,Y 261.759,Z 535.54,A -85,B 0,C 180,E1 -18079.95,E2 -18079.95} C_VEL
LIN {X 0,Y 261.336,Z 540.266,A -85,B 0,C 180,E1 -18082.273,E2 -18082.273} C_VEL
LIN {X 0,Y 261.157,Z 543.992,A -85,B 0,C 180,E1 -18084.693,E2 -18084.693} C_VEL
LIN {X 0,Y 261.145,Z 546.421,A -85,B 0,C 180,E1 -18086.915,E2 -18086.915} C_VEL
LIN {X 0,Y 261.164,Z 547.615,A -85,B 0,C 180,E1 -18088.459,E2 -18088.459} C_VEL
LIN {X 0,Y 261.175,Z 548.361,A -85,B 0,C 180,E1 -18090.001,E2 -18090.001} C_VEL
LIN {X 0,Y 261.141,Z 548.704,A -85,B 0,C 180,E1 -18091.543,E2 -18091.543} C_VEL
LIN {X 0,Y 261.106,Z 548.659,A -85,B 0,C 180,E1 -18093.087,E2 -18093.087} C_VEL
LIN {X 0,Y 261.086,Z 547.979,A -85,B 0,C 180,E1 -18095.138,E2 -18095.138} C_VEL
LIN {X 0,Y 261.35,Z 546.119,A -85,B 0,C 180,E1 -18097.728,E2 -18097.728} C_VEL
LIN {X 0,Y 261.92,Z 543.474,A -85,B 0,C 180,E1 -18100.045,E2 -18100.045} C_VEL
LIN {X 0,Y 262.791,Z 539.834,A -85,B 0,C 180,E1 -18102.355,E2 -18102.355} C_VEL
LIN {X 0,Y 264.137,Z 535.108,A -85,B 0,C 180,E1 -18104.642,E2 -18104.642} C_VEL
LIN {X 0,Y 266.251,Z 528.035,A -85,B 0,C 180,E1 -18107.275,E2 -18107.275} C_VEL
LIN {X 0,Y 268.349,Z 520.148,A -85,B 0,C 180,E1 -18109.575,E2 -18109.575} C_VEL
LIN {X 0,Y 270.873,Z 510.825,A -85,B 0,C 180,E1 -18111.699,E2 -18111.699} C_VEL
LIN {X 0,Y 273.407,Z 500.974,A -85,B 0,C 180,E1 -18113.481,E2 -18113.481} C_VEL
LIN {X 0,Y 275.921,Z 489.94,A -85,B 0,C 180,E1 -18115.053,E2 -18115.053} C_VEL
LIN {X 0,Y 278.398,Z 477.392,A -85,B 0,C 180,E1 -18116.42,E2 -18116.42} C_VEL
LIN {X 0,Y 280.387,Z 464.967,A -85,B 0,C 180,E1 -18117.425,E2 -18117.425} C_VEL
LIN {X 0,Y 281.965,Z 451.714,A -85,B 0,C 180,E1 -18118.166,E2 -18118.166} C_VEL
LIN {X 0,Y 282.834,Z 438.287,A -85,B 0,C 180,E1 -18118.649,E2 -18118.649} C_VEL
LIN {X 0,Y 284.638,Z 387.168,A -85,B 0,C 180,E1 -18119.932,E2 -18119.932} C_VEL
LIN {X 0,Y 281.027,Z 365.447,A -85,B 0,C 180,E1 -18121.086,E2 -18121.086} C_VEL
LIN {X 0,Y 279.934,Z 360.515,A -85,B 0,C 180,E1 -18121.394,E2 -18121.394} C_VEL
LIN {X 0,Y 273.898,Z 347.295,A -85,B 0,C 180,E1 -18122.709,E2 -18122.709} C_VEL
LIN {X 0,Y 267.612,Z 334.715,A -85,B 0,C 180,E1 -18124.146,E2 -18124.146} C_VEL
LIN {X 0,Y 265.611,Z 326.466,A -85,B 0,C 180,E1 -18127.487,E2 -18127.487} C_VEL
LIN {X 0,Y 263.134,Z 317.71,A -85,B 0,C 180,E1 -18131.408,E2 -18131.408} C_VEL
LIN {X 0,Y 263.125,Z 317.711,A -85,B 0,C 180,E1 -18136.016,E2 -18136.016} C_VEL
LIN {X 0,Y 263.107,Z 317.705,A -85,B 0,C 180,E1 -18140.127,E2 -18140.127} C_VEL
LIN {X 0,Y 263.164,Z 317.702,A -85,B 0,C 180,E1 -18144.018,E2 -18144.018} C_VEL
LIN {X 0,Y 263.134,Z 317.707,A -85,B 0,C 180,E1 -18147.712,E2 -18147.712} C_VEL
LIN {X 0,Y 263.203,Z 317.698,A -85,B 0,C 180,E1 -18151.783,E2 -18151.783} C_VEL
LIN {X 0,Y 263.227,Z 317.698,A -85,B 0,C 180,E1 -18155.2,E2 -18155.2} C_VEL
LIN {X 0,Y 263.265,Z 317.69,A -85,B 0,C 180,E1 -18159.693,E2 -18159.693} C_VEL
LIN {X 0,Y 263.352,Z 317.675,A -85,B 0,C 180,E1 -18164.522,E2 -18164.522} C_VEL
LIN {X 0,Y 263.356,Z 317.67,A -85,B 0,C 180,E1 -18169.233,E2 -18169.233} C_VEL
LIN {X 0,Y 263.559,Z 317.649,A -85,B 0,C 180,E1 -18172.338,E2 -18172.338} C_VEL
LIN {X 0,Y 263.751,Z 317.614,A -85,B 0,C 180,E1 -18178.473,E2 -18178.473} C_VEL
LIN {X 0,Y 263.751,Z 317.626,A -85,B 0,C 180,E1 -18181.527,E2 -18181.527} C_VEL
LIN {X 0,Y 263.573,Z 317.64,A -85,B 0,C 180,E1 -18187.661,E2 -18187.661} C_VEL
LIN {X 0,Y 263.374,Z 317.673,A -85,B 0,C 180,E1 -18190.765,E2 -18190.765} C_VEL
LIN {X 0,Y 263.351,Z 317.677,A -85,B 0,C 180,E1 -18195.478,E2 -18195.478} C_VEL
LIN {X 0,Y 263.263,Z 317.684,A -85,B 0,C 180,E1 -18200.306,E2 -18200.306} C_VEL
LIN {X 0,Y 263.193,Z 317.693,A -85,B 0,C 180,E1 -18205.293,E2 -18205.293} C_VEL
LIN {X 0,Y 263.166,Z 317.694,A -85,B 0,C 180,E1 -18208.731,E2 -18208.731} C_VEL
LIN {X 0,Y 263.133,Z 317.7,A -85,B 0,C 180,E1 -18212.288,E2 -18212.288} C_VEL
LIN {X 0,Y 263.183,Z 317.699,A -85,B 0,C 180,E1 -18216.763,E2 -18216.763} C_VEL
LIN {X 0,Y 263.125,Z 317.711,A -85,B 0,C 180,E1 -18221.593,E2 -18221.593} C_VEL
LIN {X 0,Y 263.142,Z 317.786,A -85,B 0,C 180,E1 -18224.514,E2 -18224.514} C_VEL
LIN {X 0,Y 263.489,Z 319.247,A -85,B 0,C 180,E1 -18225.18,E2 -18225.18} C_VEL
LIN {X 0,Y 265.962,Z 323.416,A -85,B 0,C 180,E1 -18225.763,E2 -18225.763} C_VEL
LIN {X 0,Y 274.957,Z 339.332,A -85,B 0,C 180,E1 -18227.754,E2 -18227.754} C_VEL
LIN {X 0,Y 282.924,Z 355.693,A -85,B 0,C 180,E1 -18229.439,E2 -18229.439} C_VEL
LIN {X 0,Y 285.539,Z 361.879,A -85,B 0,C 180,E1 -18229.989,E2 -18229.989} C_VEL
LIN {X 0,Y 282.991,Z 426.44,A -85,B 0,C 180,E1 -18231.62,E2 -18231.62} C_VEL
LIN {X 0,Y 281.878,Z 439.832,A -85,B 0,C 180,E1 -18232.236,E2 -18232.236} C_VEL
LIN {X 0,Y 280.658,Z 450.379,A -85,B 0,C 180,E1 -18232.947,E2 -18232.947} C_VEL
LIN {X 0,Y 279.054,Z 462.031,A -85,B 0,C 180,E1 -18234.006,E2 -18234.006} C_VEL
LIN {X 0,Y 277.146,Z 472.439,A -85,B 0,C 180,E1 -18235.21,E2 -18235.21} C_VEL
LIN {X 0,Y 274.781,Z 483.555,A -85,B 0,C 180,E1 -18236.859,E2 -18236.859} C_VEL
LIN {X 0,Y 272.358,Z 493.187,A -85,B 0,C 180,E1 -18238.647,E2 -18238.647} C_VEL
LIN {X 0,Y 269.843,Z 502.262,A -85,B 0,C 180,E1 -18240.768,E2 -18240.768} C_VEL
LIN {X 0,Y 267.856,Z 509.021,A -85,B 0,C 180,E1 -18242.751,E2 -18242.751} C_VEL
LIN {X 0,Y 266.009,Z 515.13,A -85,B 0,C 180,E1 -18244.993,E2 -18244.993} C_VEL
LIN {X 0,Y 264.421,Z 520.128,A -85,B 0,C 180,E1 -18247.331,E2 -18247.331} C_VEL
LIN {X 0,Y 263.173,Z 523.948,A -85,B 0,C 180,E1 -18249.686,E2 -18249.686} C_VEL
LIN {X 0,Y 262.492,Z 525.902,A -85,B 0,C 180,E1 -18251.259,E2 -18251.259} C_VEL
LIN {X 0,Y 261.999,Z 527.42,A -85,B 0,C 180,E1 -18252.838,E2 -18252.838} C_VEL
LIN {X 0,Y 261.468,Z 528.933,A -85,B 0,C 180,E1 -18255.385,E2 -18255.385} C_VEL
LIN {X 0,Y 261.154,Z 529.37,A -85,B 0,C 180,E1 -18257.567,E2 -18257.567} C_VEL
LIN {X 0,Y 260.974,Z 529.221,A -85,B 0,C 180,E1 -18259.134,E2 -18259.134} C_VEL
LIN {X 0,Y 261.014,Z 528.632,A -85,B 0,C 180,E1 -18260.702,E2 -18260.702} C_VEL
LIN {X 0,Y 261.089,Z 527.656,A -85,B 0,C 180,E1 -18262.264,E2 -18262.264} C_VEL
LIN {X 0,Y 261.325,Z 525.759,A -85,B 0,C 180,E1 -18264.305,E2 -18264.305} C_VEL
LIN {X 0,Y 261.594,Z 522.221,A -85,B 0,C 180,E1 -18266.919,E2 -18266.919} C_VEL
LIN {X 0,Y 262.158,Z 517.957,A -85,B 0,C 180,E1 -18269.231,E2 -18269.231} C_VEL
LIN {X 0,Y 262.997,Z 511.522,A -85,B 0,C 180,E1 -18271.913,E2 -18271.913} C_VEL
LIN {X 0,Y 264.201,Z 504.448,A -85,B 0,C 180,E1 -18274.194,E2 -18274.194} C_VEL
LIN {X 0,Y 265.558,Z 495.653,A -85,B 0,C 180,E1 -18276.457,E2 -18276.457} C_VEL
LIN {X 0,Y 266.979,Z 486.635,A -85,B 0,C 180,E1 -18278.324,E2 -18278.324} C_VEL
LIN {X 0,Y 268.44,Z 476.683,A -85,B 0,C 180,E1 -18279.987,E2 -18279.987} C_VEL
LIN {X 0,Y 269.906,Z 467.143,A -85,B 0,C 180,E1 -18281.261,E2 -18281.261} C_VEL
LIN {X 0,Y 271.113,Z 457.111,A -85,B 0,C 180,E1 -18282.348,E2 -18282.348} C_VEL
LIN {X 0,Y 272.029,Z 445.293,A -85,B 0,C 180,E1 -18283.349,E2 -18283.349} C_VEL
LIN {X 0,Y 272.759,Z 432.551,A -85,B 0,C 180,E1 -18284.12,E2 -18284.12} C_VEL
LIN {X 0,Y 273.534,Z 420.5,A -85,B 0,C 180,E1 -18284.554,E2 -18284.554} C_VEL
LIN {X 0,Y 275.348,Z 351.131,A -85,B 0,C 180,E1 -18286.333,E2 -18286.333} C_VEL
LIN {X 0,Y 273.318,Z 344.042,A -85,B 0,C 180,E1 -18286.711,E2 -18286.711} C_VEL
LIN {X 0,Y 265.721,Z 323.953,A -85,B 0,C 180,E1 -18287.995,E2 -18287.995} C_VEL
LIN {X 0,Y 263.33,Z 318.193,A -85,B 0,C 180,E1 -18288.436,E2 -18288.436} C_VEL
LIN {X 0,Y 263.254,Z 317.694,A -85,B 0,C 180,E1 -18288.684,E2 -18288.684} C_VEL
LIN {X 0,Y 263.136,Z 317.707,A -85,B 0,C 180,E1 -18291.956,E2 -18291.956} C_VEL
LIN {X 0,Y 263.164,Z 317.7,A -85,B 0,C 180,E1 -18295.295,E2 -18295.295} C_VEL
LIN {X 0,Y 263.13,Z 317.707,A -85,B 0,C 180,E1 -18298.734,E2 -18298.734} C_VEL
LIN {X 0,Y 263.125,Z 317.707,A -85,B 0,C 180,E1 -18302.288,E2 -18302.288} C_VEL
LIN {X 0,Y 263.174,Z 317.704,A -85,B 0,C 180,E1 -18306.761,E2 -18306.761} C_VEL
LIN {X 0,Y 263.087,Z 317.71,A -85,B 0,C 180,E1 -18309.874,E2 -18309.874} C_VEL
LIN {X 0,Y 263.077,Z 317.705,A -85,B 0,C 180,E1 -18313.992,E2 -18313.992} C_VEL
LIN {X 0,Y 263.119,Z 317.706,A -85,B 0,C 180,E1 -18318.406,E2 -18318.406} C_VEL
LIN {X 0,Y 263.153,Z 317.696,A -85,B 0,C 180,E1 -18322.102,E2 -18322.102} C_VEL
LIN {X 0,Y 263.145,Z 317.704,A -85,B 0,C 180,E1 -18325.885,E2 -18325.885} C_VEL
LIN {X 0,Y 263.135,Z 317.697,A -85,B 0,C 180,E1 -18329.505,E2 -18329.505} C_VEL
LIN {X 0,Y 263.185,Z 317.697,A -85,B 0,C 180,E1 -18333.002,E2 -18333.002} C_VEL
LIN {X 0,Y 263.148,Z 317.702,A -85,B 0,C 180,E1 -18336.384,E2 -18336.384} C_VEL
LIN {X 0,Y 263.256,Z 317.681,A -85,B 0,C 180,E1 -18339.693,E2 -18339.693} C_VEL
LIN {X 0,Y 263.344,Z 317.68,A -85,B 0,C 180,E1 -18344.522,E2 -18344.522} C_VEL
LIN {X 0,Y 263.348,Z 317.67,A -85,B 0,C 180,E1 -18349.233,E2 -18349.233} C_VEL
LIN {X 0,Y 263.526,Z 317.655,A -85,B 0,C 180,E1 -18352.337,E2 -18352.337} C_VEL
LIN {X 0,Y 263.441,Z 317.665,A -85,B 0,C 180,E1 -18354.221,E2 -18354.221} C_VEL
LIN {X 0,Y 262.717,Z 317.759,A -85,B 0,C 180,E1 -18355.499,E2 -18355.499} C_VEL
LIN {X 0,Y 259.99,Z 318.096,A -85,B 0,C 180,E1 -18357.589,E2 -18357.589} C_VEL
LIN {X 0,Y 257.736,Z 318.37,A -85,B 0,C 180,E1 -18359.288,E2 -18359.288} C_VEL
LIN {X 0,Y 256.778,Z 318.486,A -85,B 0,C 180,E1 -18360.6,E2 -18360.6} C_VEL
LIN {X 0,Y 256.7,Z 318.494,A -85,B 0,C 180,E1 -18361.044,E2 -18361.044} C_VEL
LIN {X 0,Y 256.478,Z 318.538,A -85,B 0,C 180,E1 -18366.293,E2 -18366.293} C_VEL
LIN {X 0,Y 256.455,Z 318.53,A -85,B 0,C 180,E1 -18369.464,E2 -18369.464} C_VEL
LIN {X 0,Y 256.245,Z 318.563,A -85,B 0,C 180,E1 -18374.291,E2 -18374.291} C_VEL
LIN {X 0,Y 256.204,Z 318.567,A -85,B 0,C 180,E1 -18377.563,E2 -18377.563} C_VEL
LIN {X 0,Y 256.152,Z 318.577,A -85,B 0,C 180,E1 -18381.12,E2 -18381.12} C_VEL
LIN {X 0,Y 256.183,Z 318.574,A -85,B 0,C 180,E1 -18385.139,E2 -18385.139} C_VEL
LIN {X 0,Y 256.109,Z 318.581,A -85,B 0,C 180,E1 -18389.601,E2 -18389.601} C_VEL
LIN {X 0,Y 256.081,Z 318.588,A -85,B 0,C 180,E1 -18393.291,E2 -18393.291} C_VEL
LIN {X 0,Y 256.125,Z 318.583,A -85,B 0,C 180,E1 -18397.276,E2 -18397.276} C_VEL
LIN {X 0,Y 256.053,Z 318.593,A -85,B 0,C 180,E1 -18401.204,E2 -18401.204} C_VEL
LIN {X 0,Y 256.038,Z 318.595,A -85,B 0,C 180,E1 -18405.535,E2 -18405.535} C_VEL
LIN {X 0,Y 256.052,Z 318.589,A -85,B 0,C 180,E1 -18408.798,E2 -18408.798} C_VEL
LIN {X 0,Y 256.13,Z 318.58,A -85,B 0,C 180,E1 -18412.869,E2 -18412.869} C_VEL
LIN {X 0,Y 256.111,Z 318.634,A -85,B 0,C 180,E1 -18415.181,E2 -18415.181} C_VEL
LIN {X 0,Y 258.601,Z 329.912,A -85,B 0,C 180,E1 -18419.279,E2 -18419.279} C_VEL
LIN {X 0,Y 259.78,Z 335.795,A -85,B 0,C 180,E1 -18421.266,E2 -18421.266} C_VEL
LIN {X 0,Y 263.003,Z 345.237,A -85,B 0,C 180,E1 -18421.865,E2 -18421.865} C_VEL
LIN {X 0,Y 266.932,Z 375.556,A -85,B 0,C 180,E1 -18423.112,E2 -18423.112} C_VEL
LIN {X 0,Y 268.033,Z 385.611,A -85,B 0,C 180,E1 -18423.498,E2 -18423.498} C_VEL
LIN {X 0,Y 266.332,Z 444.663,A -85,B 0,C 180,E1 -18425.079,E2 -18425.079} C_VEL
LIN {X 0,Y 265.355,Z 458.616,A -85,B 0,C 180,E1 -18425.764,E2 -18425.764} C_VEL
LIN {X 0,Y 264.129,Z 471.101,A -85,B 0,C 180,E1 -18426.686,E2 -18426.686} C_VEL
LIN {X 0,Y 262.503,Z 483.831,A -85,B 0,C 180,E1 -18427.988,E2 -18427.988} C_VEL
LIN {X 0,Y 260.787,Z 495.149,A -85,B 0,C 180,E1 -18429.493,E2 -18429.493} C_VEL
LIN {X 0,Y 259.236,Z 505.63,A -85,B 0,C 180,E1 -18431.281,E2 -18431.281} C_VEL
LIN {X 0,Y 258.028,Z 513.715,A -85,B 0,C 180,E1 -18432.975,E2 -18432.975} C_VEL
LIN {X 0,Y 256.542,Z 522.798,A -85,B 0,C 180,E1 -18435.322,E2 -18435.322} C_VEL
LIN {X 0,Y 255.326,Z 530.097,A -85,B 0,C 180,E1 -18437.684,E2 -18437.684} C_VEL
LIN {X 0,Y 254.732,Z 535.028,A -85,B 0,C 180,E1 -18439.67,E2 -18439.67} C_VEL
LIN {X 0,Y 254.29,Z 539.808,A -85,B 0,C 180,E1 -18442.058,E2 -18442.058} C_VEL
LIN {X 0,Y 254.087,Z 543.822,A -85,B 0,C 180,E1 -18444.722,E2 -18444.722} C_VEL
LIN {X 0,Y 254.058,Z 546.058,A -85,B 0,C 180,E1 -18446.829,E2 -18446.829} C_VEL
LIN {X 0,Y 254.091,Z 547.28,A -85,B 0,C 180,E1 -18448.416,E2 -18448.416} C_VEL
LIN {X 0,Y 254.101,Z 548.064,A -85,B 0,C 180,E1 -18450.001,E2 -18450.001} C_VEL
LIN {X 0,Y 254.068,Z 548.429,A -85,B 0,C 180,E1 -18451.586,E2 -18451.586} C_VEL
LIN {X 0,Y 254.019,Z 548.405,A -85,B 0,C 180,E1 -18453.173,E2 -18453.173} C_VEL
LIN {X 0,Y 253.991,Z 547.893,A -85,B 0,C 180,E1 -18455.04,E2 -18455.04} C_VEL
LIN {X 0,Y 254.308,Z 545.951,A -85,B 0,C 180,E1 -18457.943,E2 -18457.943} C_VEL
LIN {X 0,Y 255.174,Z 542.274,A -85,B 0,C 180,E1 -18461.117,E2 -18461.117} C_VEL
LIN {X 0,Y 256.238,Z 538.327,A -85,B 0,C 180,E1 -18463.482,E2 -18463.482} C_VEL
LIN {X 0,Y 257.848,Z 533.272,A -85,B 0,C 180,E1 -18465.818,E2 -18465.818} C_VEL
LIN {X 0,Y 259.751,Z 526.945,A -85,B 0,C 180,E1 -18468.129,E2 -18468.129} C_VEL
LIN {X 0,Y 261.981,Z 519.055,A -85,B 0,C 180,E1 -18470.411,E2 -18470.411} C_VEL
LIN {X 0,Y 264.284,Z 511.042,A -85,B 0,C 180,E1 -18472.269,E2 -18472.269} C_VEL
LIN {X 0,Y 266.931,Z 501.286,A -85,B 0,C 180,E1 -18474.086,E2 -18474.086} C_VEL
LIN {X 0,Y 269.528,Z 490.444,A -85,B 0,C 180,E1 -18475.69,E2 -18475.69} C_VEL
LIN {X 0,Y 272.091,Z 478.091,A -85,B 0,C 180,E1 -18477.081,E2 -18477.081} C_VEL
LIN {X 0,Y 274.157,Z 465.995,A -85,B 0,C 180,E1 -18478.102,E2 -18478.102} C_VEL
LIN {X 0,Y 275.778,Z 453.451,A -85,B 0,C 180,E1 -18478.856,E2 -18478.856} C_VEL
LIN {X 0,Y 276.763,Z 440.204,A -85,B 0,C 180,E1 -18479.376,E2 -18479.376} C_VEL
LIN {X 0,Y 278.781,Z 388.475,A -85,B 0,C 180,E1 -18480.696,E2 -18480.696} C_VEL
LIN {X 0,Y 274.991,Z 365.732,A -85,B 0,C 180,E1 -18481.956,E2 -18481.956} C_VEL
LIN {X 0,Y 273.905,Z 362.15,A -85,B 0,C 180,E1 -18482.234,E2 -18482.234} C_VEL
LIN {X 0,Y 268.445,Z 350.409,A -85,B 0,C 180,E1 -18483.471,E2 -18483.471} C_VEL
LIN {X 0,Y 262.055,Z 337.936,A -85,B 0,C 180,E1 -18484.973,E2 -18484.973} C_VEL
LIN {X 0,Y 260.376,Z 334.38,A -85,B 0,C 180,E1 -18485.405,E2 -18485.405} C_VEL
LIN {X 0,Y 258.104,Z 325.665,A -85,B 0,C 180,E1 -18489.152,E2 -18489.152} C_VEL
LIN {X 0,Y 256.049,Z 318.588,A -85,B 0,C 180,E1 -18492.499,E2 -18492.499} C_VEL
LIN {X 0,Y 256.063,Z 318.585,A -85,B 0,C 180,E1 -18496.673,E2 -18496.673} C_VEL
LIN {X 0,Y 256.073,Z 318.585,A -85,B 0,C 180,E1 -18500.858,E2 -18500.858} C_VEL
LIN {X 0,Y 256.131,Z 318.573,A -85,B 0,C 180,E1 -18502.867,E2 -18502.867} C_VEL
LIN {X 0,Y 256.069,Z 318.58,A -85,B 0,C 180,E1 -18506.707,E2 -18506.707} C_VEL
LIN {X 0,Y 256.115,Z 318.577,A -85,B 0,C 180,E1 -18510.4,E2 -18510.4} C_VEL
LIN {X 0,Y 256.19,Z 318.572,A -85,B 0,C 180,E1 -18514.861,E2 -18514.861} C_VEL
LIN {X 0,Y 256.168,Z 318.575,A -85,B 0,C 180,E1 -18519.105,E2 -18519.105} C_VEL
LIN {X 0,Y 256.301,Z 318.555,A -85,B 0,C 180,E1 -18524.085,E2 -18524.085} C_VEL
LIN {X 0,Y 256.298,Z 318.551,A -85,B 0,C 180,E1 -18528.933,E2 -18528.933} C_VEL
LIN {X 0,Y 256.516,Z 318.528,A -85,B 0,C 180,E1 -18532.126,E2 -18532.126} C_VEL
LIN {X 0,Y 256.498,Z 318.528,A -85,B 0,C 180,E1 -18536.858,E2 -18536.858} C_VEL
LIN {X 0,Y 256.758,Z 318.489,A -85,B 0,C 180,E1 -18540,E2 -18540} C_VEL
LIN {X 0,Y 256.498,Z 318.519,A -85,B 0,C 180,E1 -18543.141,E2 -18543.141} C_VEL
LIN {X 0,Y 256.54,Z 318.516,A -85,B 0,C 180,E1 -18547.873,E2 -18547.873} C_VEL
LIN {X 0,Y 256.31,Z 318.552,A -85,B 0,C 180,E1 -18551.066,E2 -18551.066} C_VEL
LIN {X 0,Y 256.3,Z 318.552,A -85,B 0,C 180,E1 -18555.915,E2 -18555.915} C_VEL
LIN {X 0,Y 256.163,Z 318.568,A -85,B 0,C 180,E1 -18560.895,E2 -18560.895} C_VEL
LIN {X 0,Y 256.171,Z 318.567,A -85,B 0,C 180,E1 -18565.13,E2 -18565.13} C_VEL
LIN {X 0,Y 256.104,Z 318.581,A -85,B 0,C 180,E1 -18569.601,E2 -18569.601} C_VEL
LIN {X 0,Y 256.068,Z 318.586,A -85,B 0,C 180,E1 -18573.293,E2 -18573.293} C_VEL
LIN {X 0,Y 256.115,Z 318.576,A -85,B 0,C 180,E1 -18577.27,E2 -18577.27} C_VEL
LIN {X 0,Y 256.055,Z 318.589,A -85,B 0,C 180,E1 -18581.203,E2 -18581.203} C_VEL
LIN {X 0,Y 256.074,Z 318.733,A -85,B 0,C 180,E1 -18583.45,E2 -18583.45} C_VEL
LIN {X 0,Y 256.361,Z 319.789,A -85,B 0,C 180,E1 -18583.895,E2 -18583.895} C_VEL
LIN {X 0,Y 257.787,Z 322.398,A -85,B 0,C 180,E1 -18584.259,E2 -18584.259} C_VEL
LIN {X 0,Y 264.002,Z 332.534,A -85,B 0,C 180,E1 -18585.735,E2 -18585.735} C_VEL
LIN {X 0,Y 272.244,Z 347.828,A -85,B 0,C 180,E1 -18587.605,E2 -18587.605} C_VEL
LIN {X 0,Y 278.644,Z 361.546,A -85,B 0,C 180,E1 -18589.006,E2 -18589.006} C_VEL
LIN {X 0,Y 279.604,Z 363.917,A -85,B 0,C 180,E1 -18589.218,E2 -18589.218} C_VEL
LIN {X 0,Y 277.073,Z 426.275,A -85,B 0,C 180,E1 -18590.82,E2 -18590.82} C_VEL
LIN {X 0,Y 275.911,Z 439.803,A -85,B 0,C 180,E1 -18591.445,E2 -18591.445} C_VEL
LIN {X 0,Y 274.73,Z 449.846,A -85,B 0,C 180,E1 -18592.124,E2 -18592.124} C_VEL
LIN {X 0,Y 273.058,Z 461.607,A -85,B 0,C 180,E1 -18593.195,E2 -18593.195} C_VEL
LIN {X 0,Y 270.902,Z 472.913,A -85,B 0,C 180,E1 -18594.516,E2 -18594.516} C_VEL
LIN {X 0,Y 268.434,Z 483.979,A -85,B 0,C 180,E1 -18596.195,E2 -18596.195} C_VEL
LIN {X 0,Y 265.831,Z 493.858,A -85,B 0,C 180,E1 -18598.078,E2 -18598.078} C_VEL
LIN {X 0,Y 263.49,Z 501.908,A -85,B 0,C 180,E1 -18599.992,E2 -18599.992} C_VEL
LIN {X 0,Y 261.082,Z 509.706,A -85,B 0,C 180,E1 -18602.331,E2 -18602.331} C_VEL
LIN {X 0,Y 258.778,Z 516.836,A -85,B 0,C 180,E1 -18605.105,E2 -18605.105} C_VEL
LIN {X 0,Y 257.214,Z 521.524,A -85,B 0,C 180,E1 -18607.509,E2 -18607.509} C_VEL
LIN {X 0,Y 256.362,Z 523.984,A -85,B 0,C 180,E1 -18609.121,E2 -18609.121} C_VEL
LIN {X 0,Y 255.613,Z 525.975,A -85,B 0,C 180,E1 -18610.735,E2 -18610.735} C_VEL
LIN {X 0,Y 255.042,Z 527.538,A -85,B 0,C 180,E1 -18612.354,E2 -18612.354} C_VEL
LIN {X 0,Y 254.41,Z 529.218,A -85,B 0,C 180,E1 -18615.209,E2 -18615.209} C_VEL
LIN {X 0,Y 254.091,Z 529.621,A -85,B 0,C 180,E1 -18617.215,E2 -18617.215} C_VEL
LIN {X 0,Y 253.899,Z 529.524,A -85,B 0,C 180,E1 -18618.827,E2 -18618.827} C_VEL
LIN {X 0,Y 253.898,Z 528.987,A -85,B 0,C 180,E1 -18620.439,E2 -18620.439} C_VEL
LIN {X 0,Y 253.973,Z 528.045,A -85,B 0,C 180,E1 -18622.046,E2 -18622.046} C_VEL
LIN {X 0,Y 254.238,Z 525.975,A -85,B 0,C 180,E1 -18624.36,E2 -18624.36} C_VEL
LIN {X 0,Y 254.508,Z 522.75,A -85,B 0,C 180,E1 -18626.833,E2 -18626.833} C_VEL
LIN {X 0,Y 255.059,Z 518.567,A -85,B 0,C 180,E1 -18629.21,E2 -18629.21} C_VEL
LIN {X 0,Y 255.915,Z 512.218,A -85,B 0,C 180,E1 -18631.966,E2 -18631.966} C_VEL
LIN {X 0,Y 257.124,Z 505.285,A -85,B 0,C 180,E1 -18634.31,E2 -18634.31} C_VEL
LIN {X 0,Y 258.542,Z 496.611,A -85,B 0,C 180,E1 -18636.633,E2 -18636.633} C_VEL
LIN {X 0,Y 259.99,Z 487.731,A -85,B 0,C 180,E1 -18638.549,E2 -18638.549} C_VEL
LIN {X 0,Y 261.491,Z 477.973,A -85,B 0,C 180,E1 -18640.256,E2 -18640.256} C_VEL
LIN {X 0,Y 263.185,Z 467.184,A -85,B 0,C 180,E1 -18641.747,E2 -18641.747} C_VEL
LIN {X 0,Y 264.439,Z 457.095,A -85,B 0,C 180,E1 -18642.86,E2 -18642.86} C_VEL
LIN {X 0,Y 265.383,Z 445.193,A -85,B 0,C 180,E1 -18643.885,E2 -18643.885} C_VEL
LIN {X 0,Y 266.1,Z 433.208,A -85,B 0,C 180,E1 -18644.628,E2 -18644.628} C_VEL
LIN {X 0,Y 266.948,Z 419.912,A -85,B 0,C 180,E1 -18645.117,E2 -18645.117} C_VEL
LIN {X 0,Y 268.838,Z 352.188,A -85,B 0,C 180,E1 -18646.885,E2 -18646.885} C_VEL
LIN {X 0,Y 264.065,Z 338.076,A -85,B 0,C 180,E1 -18647.743,E2 -18647.743} C_VEL
LIN {X 0,Y 258.312,Z 323.724,A -85,B 0,C 180,E1 -18648.745,E2 -18648.745} C_VEL
LIN {X 0,Y 256.26,Z 319.009,A -85,B 0,C 180,E1 -18649.103,E2 -18649.103} C_VEL
LIN {X 0,Y 256.2,Z 318.572,A -85,B 0,C 180,E1 -18649.163,E2 -18649.163} C_VEL
LIN {X 0,Y 256.074,Z 318.588,A -85,B 0,C 180,E1 -18652.595,E2 -18652.595} C_VEL
LIN {X 0,Y 256.096,Z 318.581,A -85,B 0,C 180,E1 -18656.044,E2 -18656.044} C_VEL
LIN {X 0,Y 256.052,Z 318.586,A -85,B 0,C 180,E1 -18659.606,E2 -18659.606} C_VEL
LIN {X 0,Y 256.063,Z 318.588,A -85,B 0,C 180,E1 -18663.292,E2 -18663.292} C_VEL
LIN {X 0,Y 256.108,Z 318.579,A -85,B 0,C 180,E1 -18667.269,E2 -18667.269} C_VEL
LIN {X 0,Y 256.014,Z 318.595,A -85,B 0,C 180,E1 -18671.21,E2 -18671.21} C_VEL
LIN {X 0,Y 256.032,Z 318.59,A -85,B 0,C 180,E1 -18675.534,E2 -18675.534} C_VEL
LIN {X 0,Y 256.049,Z 318.589,A -85,B 0,C 180,E1 -18678.796,E2 -18678.796} C_VEL
LIN {X 0,Y 256.123,Z 318.573,A -85,B 0,C 180,E1 -18682.866,E2 -18682.866} C_VEL
LIN {X 0,Y 256.062,Z 318.585,A -85,B 0,C 180,E1 -18686.707,E2 -18686.707} C_VEL
LIN {X 0,Y 256.098,Z 318.571,A -85,B 0,C 180,E1 -18690.399,E2 -18690.399} C_VEL
LIN {X 0,Y 256.165,Z 318.574,A -85,B 0,C 180,E1 -18694.87,E2 -18694.87} C_VEL
LIN {X 0,Y 256.156,Z 318.566,A -85,B 0,C 180,E1 -18699.104,E2 -18699.104} C_VEL
LIN {X 0,Y 256.293,Z 318.561,A -85,B 0,C 180,E1 -18704.085,E2 -18704.085} C_VEL
LIN {X 0,Y 256.29,Z 318.548,A -85,B 0,C 180,E1 -18708.933,E2 -18708.933} C_VEL
LIN {X 0,Y 256.488,Z 318.529,A -85,B 0,C 180,E1 -18712.126,E2 -18712.126} C_VEL
LIN {X 0,Y 256.489,Z 318.532,A -85,B 0,C 180,E1 -18716.859,E2 -18716.859} C_VEL
LIN {X 0,Y 256.75,Z 318.491,A -85,B 0,C 180,E1 -18720,E2 -18720} C_VEL
LIN {X 0,Y 256.7,Z 318.494,A -85,B 0,C 180,E1 -18721.044,E2 -18721.044} C_VEL
LIN {X 0,Y 256,Z 318.589,A -85,B 0,C 180,E1 -18722.35,E2 -18722.35} C_VEL
LIN {X 0,Y 253.028,Z 318.966,A -85,B 0,C 180,E1 -18724.474,E2 -18724.474} C_VEL
LIN {X 0,Y 250.542,Z 319.277,A -85,B 0,C 180,E1 -18726.204,E2 -18726.204} C_VEL
LIN {X 0,Y 249.523,Z 319.4,A -85,B 0,C 180,E1 -18727.55,E2 -18727.55} C_VEL
LIN {X 0,Y 249.467,Z 319.408,A -85,B 0,C 180,E1 -18728.005,E2 -18728.005} C_VEL
LIN {X 0,Y 249.246,Z 319.424,A -85,B 0,C 180,E1 -18731.384,E2 -18731.384} C_VEL
LIN {X 0,Y 249.212,Z 319.443,A -85,B 0,C 180,E1 -18736.504,E2 -18736.504} C_VEL
LIN {X 0,Y 249.082,Z 319.455,A -85,B 0,C 180,E1 -18741.519,E2 -18741.519} C_VEL
LIN {X 0,Y 249.126,Z 319.451,A -85,B 0,C 180,E1 -18745.483,E2 -18745.483} C_VEL
LIN {X 0,Y 249.079,Z 319.461,A -85,B 0,C 180,E1 -18748.994,E2 -18748.994} C_VEL
LIN {X 0,Y 249.032,Z 319.465,A -85,B 0,C 180,E1 -18752.426,E2 -18752.426} C_VEL
LIN {X 0,Y 249.065,Z 319.46,A -85,B 0,C 180,E1 -18756.34,E2 -18756.34} C_VEL
LIN {X 0,Y 249.022,Z 319.466,A -85,B 0,C 180,E1 -18760.475,E2 -18760.475} C_VEL
LIN {X 0,Y 248.982,Z 319.471,A -85,B 0,C 180,E1 -18764.884,E2 -18764.884} C_VEL
LIN {X 0,Y 249.007,Z 319.47,A -85,B 0,C 180,E1 -18767.363,E2 -18767.363} C_VEL
LIN {X 0,Y 249.024,Z 319.466,A -85,B 0,C 180,E1 -18771.621,E2 -18771.621} C_VEL
LIN {X 0,Y 249.085,Z 319.474,A -85,B 0,C 180,E1 -18774.621,E2 -18774.621} C_VEL
LIN {X 0,Y 251.536,Z 330.822,A -85,B 0,C 180,E1 -18778.878,E2 -18778.878} C_VEL
LIN {X 0,Y 252.483,Z 335.325,A -85,B 0,C 180,E1 -18780.495,E2 -18780.495} C_VEL
LIN {X 0,Y 256.659,Z 347.083,A -85,B 0,C 180,E1 -18781.291,E2 -18781.291} C_VEL
LIN {X 0,Y 260.515,Z 377.272,A -85,B 0,C 180,E1 -18782.571,E2 -18782.571} C_VEL
LIN {X 0,Y 261.498,Z 386.282,A -85,B 0,C 180,E1 -18782.928,E2 -18782.928} C_VEL
LIN {X 0,Y 259.746,Z 444.201,A -85,B 0,C 180,E1 -18784.51,E2 -18784.51} C_VEL
LIN {X 0,Y 258.773,Z 457.443,A -85,B 0,C 180,E1 -18785.159,E2 -18785.159} C_VEL
LIN {X 0,Y 257.622,Z 469.638,A -85,B 0,C 180,E1 -18786.06,E2 -18786.06} C_VEL
LIN {X 0,Y 256.137,Z 481.098,A -85,B 0,C 180,E1 -18787.198,E2 -18787.198} C_VEL
LIN {X 0,Y 254.302,Z 492.87,A -85,B 0,C 180,E1 -18788.733,E2 -18788.733} C_VEL
LIN {X 0,Y 252.676,Z 503.467,A -85,B 0,C 180,E1 -18790.503,E2 -18790.503} C_VEL
LIN {X 0,Y 251.159,Z 512.997,A -85,B 0,C 180,E1 -18792.495,E2 -18792.495} C_VEL
LIN {X 0,Y 249.646,Z 522.163,A -85,B 0,C 180,E1 -18794.907,E2 -18794.907} C_VEL
LIN {X 0,Y 248.36,Z 529.527,A -85,B 0,C 180,E1 -18797.333,E2 -18797.333} C_VEL
LIN {X 0,Y 247.723,Z 534.515,A -85,B 0,C 180,E1 -18799.374,E2 -18799.374} C_VEL
LIN {X 0,Y 247.219,Z 539.347,A -85,B 0,C 180,E1 -18801.829,E2 -18801.829} C_VEL
LIN {X 0,Y 247.056,Z 541.953,A -85,B 0,C 180,E1 -18803.467,E2 -18803.467} C_VEL
LIN {X 0,Y 246.971,Z 544.041,A -85,B 0,C 180,E1 -18805.104,E2 -18805.104} C_VEL
LIN {X 0,Y 246.955,Z 545.694,A -85,B 0,C 180,E1 -18806.738,E2 -18806.738} C_VEL
LIN {X 0,Y 247.019,Z 546.94,A -85,B 0,C 180,E1 -18808.371,E2 -18808.371} C_VEL
LIN {X 0,Y 247.028,Z 547.767,A -85,B 0,C 180,E1 -18810.001,E2 -18810.001} C_VEL
LIN {X 0,Y 246.997,Z 548.154,A -85,B 0,C 180,E1 -18811.631,E2 -18811.631} C_VEL
LIN {X 0,Y 246.916,Z 548.151,A -85,B 0,C 180,E1 -18813.264,E2 -18813.264} C_VEL
LIN {X 0,Y 246.914,Z 547.739,A -85,B 0,C 180,E1 -18814.982,E2 -18814.982} C_VEL
LIN {X 0,Y 247.009,Z 546.991,A -85,B 0,C 180,E1 -18816.536,E2 -18816.536} C_VEL
LIN {X 0,Y 247.26,Z 545.784,A -85,B 0,C 180,E1 -18818.171,E2 -18818.171} C_VEL
